  MoveL (T15717) to (119.32, 120.67, 17.1) mm, rotated rx 180 ry 0 rz -180 deg; joints [1.326, 66.029, -27.799, 2.142, -38.249, -1.682]
  Call Extruder 0.59936
  MoveL (T15718) to (105.47, 106.82, 17.1) mm, rotated rx 180 ry 0 rz -180 deg; joints [1.326, 66.029, -27.799, 2.142, -38.249, -1.682]
  Call Extruder 0.0152
  MoveL (T15719) to (105.47, 107.32, 17.1) mm, rotated rx 180 ry 0 rz -180 deg; joints [1.326, 66.029, -27.799, 2.142, -38.249, -1.682]
  Call Extruder 0.00328
  MoveL (T15720) to (105.49, 107.42, 17.1) mm, rotated rx 180 ry 0 rz -180 deg; joints [1.326, 66.029, -27.799, 2.142, -38.249, -1.682]
  Call Extruder 0.58584
  MoveL (T15721) to (119.03, 120.96, 17.1) mm, rotated rx 180 ry 0 rz -180 deg; joints [1.326, 66.029, -27.799, 2.142, -38.249, -1.682]
  Call Extruder 0.0086
  MoveL (T15722) to (118.83, 121.16, 17.1) mm, rotated rx 180 ry 0 rz -180 deg; joints [1.326, 66.029, -27.799, 2.142, -38.249, -1.682]
  Call Extruder 0.00554
  MoveL (T15723) to (118.65, 121.16, 17.1) mm, rotated rx 180 ry 0 rz -180 deg; joints [1.326, 66.029, -27.799, 2.142, -38.249, -1.682]
  Call Extruder 0.55945
  MoveL (T15724) to (105.72, 108.23, 17.1) mm, rotated rx 180 ry 0 rz -180 deg; joints [1.326, 66.029, -27.799, 2.142, -38.249, -1.682]
  Call Extruder 0.04056
  MoveL (T15725) to (106.33, 109.41, 17.1) mm, rotated rx 180 ry 0 rz -180 deg; joints [1.326, 66.029, -27.799, 2.142, -38.249, -1.682]
  Call Extruder 0.50836
  MoveL (T15726) to (118.07, 121.16, 17.1) mm, rotated rx 180 ry 0 rz -180 deg; joints [1.323, 66.013, -27.77, 2.137, -38.263, -1.678]
  Call Extruder 0.0177
  MoveL (T15727) to (117.49, 121.16, 17.1) mm, rotated rx 180 ry 0 rz -180 deg; joints [1.323, 66.013, -27.77, 2.137, -38.263, -1.678]
  Call Extruder 0.45726
  MoveL (T15728) to (106.93, 110.59, 17.1) mm, rotated rx 180 ry 0 rz -180 deg; joints [1.323, 66.013, -27.77, 2.137, -38.263, -1.678]
  Call Extruder 0.04056
  MoveL (T15729) to (107.53, 111.77, 17.1) mm, rotated rx 180 ry 0 rz -180 deg; joints [1.323, 66.013, -27.77, 2.137, -38.263, -1.678]
  Call Extruder 0.40616
  MoveL (T15730) to (116.92, 121.16, 17.1) mm, rotated rx 180 ry 0 rz -180 deg; joints [1.321, 66.248, -28.211, 2.143, -38.056, -1.688]
  Call Extruder 0.0177
  MoveL (T15731) to (116.34, 121.16, 17.1) mm, rotated rx 180 ry 0 rz -180 deg; joints [1.321, 66.248, -28.211, 2.143, -38.056, -1.688]
  Call Extruder 0.35507
  MoveL (T15732) to (108.13, 112.95, 17.1) mm, rotated rx 180 ry 0 rz -180 deg; joints [1.321, 66.248, -28.211, 2.143, -38.056, -1.688]
  Call Extruder 0.03441
  MoveL (T15733) to (108.64, 113.95, 17.1) mm, rotated rx 180 ry 0 rz -180 deg; joints [1.321, 66.248, -28.211, 2.143, -38.056, -1.688]
  Call Extruder 0.00268
  MoveL (T15734) to (108.56, 113.95, 17.1) mm, rotated rx 180 ry 0 rz -180 deg; joints [1.321, 66.248, -28.211, 2.143, -38.056, -1.688]
  Call Extruder 0.31171
  MoveL (T15735) to (115.76, 121.16, 17.1) mm, rotated rx 180 ry 0 rz -180 deg; joints [1.402, 70.427, -36.068, 2.484, -34.384, -2.05]
  Call Extruder 0.0177
  MoveL (T15736) to (115.18, 121.16, 17.1) mm, rotated rx 180 ry 0 rz -180 deg; joints [1.402, 70.427, -36.068, 2.484, -34.384, -2.05]
  Call Extruder 0.31171
  MoveL (T15737) to (107.98, 113.95, 17.1) mm, rotated rx 180 ry 0 rz -180 deg; joints [1.402, 70.427, -36.068, 2.484, -34.384, -2.05]
  Call Extruder 0.01315
  MoveL (T15738) to (107.55, 113.95, 17.1) mm, rotated rx 180 ry 0 rz -180 deg; joints [1.402, 70.427, -36.068, 2.484, -34.384, -2.05]
  Call Extruder 0.00328
  MoveL (T15739) to (107.46, 114.01, 17.1) mm, rotated rx 180 ry 0 rz -180 deg; joints [1.402, 70.427, -36.068, 2.484, -34.384, -2.05]
  Call Extruder 0.30914
  MoveL (T15740) to (114.6, 121.16, 17.1) mm, rotated rx 180 ry 0 rz -180 deg; joints [1.402, 70.427, -36.068, 2.484, -34.384, -2.05]
  Call Extruder 0.0177
  MoveL (T15741) to (114.02, 121.16, 17.1) mm, rotated rx 180 ry 0 rz -180 deg; joints [1.402, 70.427, -36.068, 2.484, -34.384, -2.05]
  Call Extruder 0.29663
  MoveL (T15742) to (107.17, 114.3, 17.1) mm, rotated rx 180 ry 0 rz -180 deg; joints [1.402, 70.427, -36.068, 2.484, -34.384, -2.05]
  Call Extruder 0.01252
  MoveL (T15743) to (106.88, 114.59, 17.1) mm, rotated rx 180 ry 0 rz -180 deg; joints [1.402, 70.427, -36.068, 2.484, -34.384, -2.05]
  Call Extruder 0.28411
  MoveL (T15744) to (113.44, 121.16, 17.1) mm, rotated rx 180 ry 0 rz -180 deg; joints [1.396, 71.177, -37.479, 2.515, -33.723, -2.092]
  Call Extruder 0.0177
  MoveL (T15745) to (112.87, 121.16, 17.1) mm, rotated rx 180 ry 0 rz -180 deg; joints [1.396, 71.177, -37.479, 2.515, -33.723, -2.092]
  Call Extruder 0.2716
  MoveL (T15746) to (106.59, 114.88, 17.1) mm, rotated rx 180 ry 0 rz -180 deg; joints [1.396, 71.177, -37.479, 2.515, -33.723, -2.092]
  Call Extruder 0.01252
  MoveL (T15747) to (106.3, 115.17, 17.1) mm, rotated rx 180 ry 0 rz -180 deg; joints [3.316, 66.49, -28.667, 5.398, -37.947, -4.261]
  Call Extruder 0.25908
  MoveL (T15748) to (112.29, 121.16, 17.1) mm, rotated rx 180 ry 0 rz -180 deg; joints [3.316, 66.49, -28.667, 5.398, -37.947, -4.261]
  Call Extruder 0.0177
  MoveL (T15749) to (111.71, 121.16, 17.1) mm, rotated rx 180 ry 0 rz -180 deg; joints [2.938, 66.441, -28.574, 4.78, -37.964, -3.772]
  Call Extruder 0.24657
  MoveL (T15750) to (106.01, 115.46, 17.1) mm, rotated rx 180 ry 0 rz -180 deg; joints [2.938, 66.441, -28.574, 4.78, -37.964, -3.772]
  Call Extruder 0.01252
  MoveL (T15751) to (105.72, 115.75, 17.1) mm, rotated rx 180 ry 0 rz -180 deg; joints [3.295, 67.406, -30.389, 5.461, -37.143, -4.358]
  Call Extruder 0.23405
  MoveL (T15752) to (111.13, 121.16, 17.1) mm, rotated rx 180 ry 0 rz -180 deg; joints [3.295, 67.406, -30.389, 5.461, -37.143, -4.358]
  Call Extruder 0.0177
  MoveL (T15753) to (110.55, 121.16, 17.1) mm, rotated rx 180 ry 0 rz -180 deg; joints [3.288, 67.704, -30.949, 5.483, -36.882, -4.391]
  Call Extruder 0.21634
  MoveL (T15754) to (105.55, 116.16, 17.1) mm, rotated rx 180 ry 0 rz -180 deg; joints [3.288, 67.704, -30.949, 5.483, -36.882, -4.391]
  Call Extruder 0.0177
  MoveL (T15755) to (105.55, 116.73, 17.1) mm, rotated rx 180 ry 0 rz -180 deg; joints [1.879, 71.218, -37.556, 3.388, -33.708, -2.819]
  Call Extruder 0.19131
  MoveL (T15756) to (109.97, 121.16, 17.1) mm, rotated rx 180 ry 0 rz -180 deg; joints [1.879, 71.218, -37.556, 3.388, -33.708, -2.819]
  Call Extruder 0.0177
  MoveL (T15757) to (109.4, 121.16, 17.1) mm, rotated rx 180 ry 0 rz -180 deg; joints [1.879, 71.218, -37.556, 3.388, -33.708, -2.819]
  Call Extruder 0.16628
  MoveL (T15758) to (105.55, 117.31, 17.1) mm, rotated rx 180 ry 0 rz -180 deg; joints [1.763, 71.207, -37.535, 3.177, -33.712, -2.644]
  Call Extruder 0.0177
  MoveL (T15759) to (105.55, 117.89, 17.1) mm, rotated rx 180 ry 0 rz -180 deg; joints [1.763, 71.207, -37.535, 3.177, -33.712, -2.644]
  Call Extruder 0.14125
  MoveL (T15760) to (108.82, 121.16, 17.1) mm, rotated rx 180 ry 0 rz -180 deg; joints [1.405, 70.111, -35.474, 2.471, -34.662, -2.033]
  Call Extruder 0.0177
  MoveL (T15761) to (108.24, 121.16, 17.1) mm, rotated rx 180 ry 0 rz -180 deg; joints [1.405, 70.111, -35.474, 2.471, -34.662, -2.033]
  Call Extruder 0.11622
  MoveL (T15762) to (105.55, 118.47, 17.1) mm, rotated rx 180 ry 0 rz -180 deg; joints [1.405, 70.111, -35.474, 2.471, -34.662, -2.033]
  Call Extruder 0.0177
  MoveL (T15763) to (105.55, 119.05, 17.1) mm, rotated rx 180 ry 0 rz -180 deg; joints [1.408, 69.782, -34.856, 2.458, -34.951, -2.015]
  Call Extruder 0.09119
  MoveL (T15764) to (107.66, 121.16, 17.1) mm, rotated rx 180 ry 0 rz -180 deg; joints [2.818, 66.427, -28.547, 4.584, -37.969, -3.616]
  Call Extruder 0.0177
  MoveL (T15765) to (107.08, 121.16, 17.1) mm, rotated rx 180 ry 0 rz -180 deg; joints [2.44, 66.386, -28.47, 3.966, -37.982, -3.128]
  Call Extruder 0.06616
  MoveL (T15766) to (105.55, 119.63, 17.1) mm, rotated rx 180 ry 0 rz -180 deg; joints [2.44, 66.386, -28.47, 3.966, -37.982, -3.128]
  Call Extruder 0.01683
  MoveL (T15767) to (105.55, 120.18, 17.1) mm, rotated rx 180 ry 0 rz -180 deg; joints [3.266, 68.664, -32.754, 5.557, -36.039, -4.499]
  Call Extruder 0.00161
  MoveL (T15768) to (105.57, 120.23, 17.1) mm, rotated rx 180 ry 0 rz -180 deg; joints [3.266, 68.664, -32.754, 5.557, -36.039, -4.499]
  Call Extruder 0.04818
  MoveL (T15769) to (106.69, 121.34, 17.1) mm, rotated rx 180 ry 0 rz -180 deg; joints [3.266, 68.664, -32.754, 5.557, -36.039, -4.499]
  Set speed (45.0 mm/s)
  Call Extruder -1.6
  MoveL (T15770) to (106.69, 121.34, 17.1) mm, rotated rx 180 ry 0 rz -180 deg; joints [3.266, 68.664, -32.754, 5.557, -36.039, -4.499]
  Set speed (120.0 mm/s)
  MoveL (T15771) to (106.69, 121.34, 17.1) mm, rotated rx 180 ry 0 rz -180 deg; joints [3.26, 68.978, -33.343, 5.583, -35.764, -4.535]
  Call Extruder -0.38
  MoveL (T15772) to (105.93, 120.58, 17.1) mm, rotated rx 180 ry 0 rz -180 deg; joints [3.26, 68.978, -33.343, 5.583, -35.764, -4.535]
  Set speed (45.0 mm/s)
  Call Extruder -0.02
  MoveL (T15773) to (105.93, 120.58, 17.1) mm, rotated rx 180 ry 0 rz -180 deg; joints [3.26, 68.978, -33.343, 5.583, -35.764, -4.535]
  Set speed (150.0 mm/s)
  MoveL (T15774) to (105.93, 120.58, 19.1) mm, rotated rx 180 ry 0 rz -180 deg; joints [2.362, 71.271, -37.657, 4.262, -33.688, -3.548]
  MoveL (T15775) to (120.54, 120.54, 19.1) mm, rotated rx 180 ry 0 rz -180 deg; joints [2.362, 71.271, -37.657, 4.262, -33.688, -3.548]
  MoveL (T15776) to (120.54, 120.54, 17.1) mm, rotated rx 180 ry 0 rz -180 deg; joints [2.362, 71.271, -37.657, 4.262, -33.688, -3.548]
  Set speed (40.0 mm/s)
  Call Extruder 2.0
  MoveL (T15777) to (120.54, 120.54, 17.1) mm, rotated rx 180 ry 0 rz -180 deg; joints [2.246, 71.257, -37.63, 4.051, -33.693, -3.372]
  Set speed (50.0 mm/s)
  MoveL (T15778) to (120.54, 120.54, 17.1) mm, rotated rx 180 ry 0 rz -180 deg; joints [2.246, 71.257, -37.63, 4.051, -33.693, -3.372]
  Call Extruder 0.02637
  MoveL (T15779) to (121.16, 121.16, 17.1) mm, rotated rx 180 ry 0 rz -180 deg; joints [2.246, 71.257, -37.63, 4.051, -33.693, -3.372]
  Set speed (45.0 mm/s)
  Call Extruder -1.6
  MoveL (T15780) to (121.16, 121.16, 17.1) mm, rotated rx 180 ry 0 rz -180 deg; joints [1.417, 68.778, -32.967, 2.421, -35.835, -1.963]
  Set speed (120.0 mm/s)
  MoveL (T15781) to (121.16, 121.16, 17.1) mm, rotated rx 180 ry 0 rz -180 deg; joints [1.417, 68.778, -32.967, 2.421, -35.835, -1.963]
  Call Extruder -0.30841
  MoveL (T15782) to (120.54, 120.54, 17.1) mm, rotated rx 180 ry 0 rz -180 deg; joints [1.42, 68.466, -32.382, 2.41, -36.109, -1.947]
  Set speed (45.0 mm/s)
  Call Extruder -0.09159
  MoveL (T15783) to (120.54, 120.54, 17.1) mm, rotated rx 180 ry 0 rz -180 deg; joints [1.42, 68.466, -32.382, 2.41, -36.109, -1.947]
  Set speed (150.0 mm/s)
  MoveL (T15784) to (120.54, 120.54, 19.1) mm, rotated rx 180 ry 0 rz -180 deg; joints [1.42, 68.466, -32.382, 2.41, -36.109, -1.947]
  MoveL (T15785) to (104.34, 103.54, 19.1) mm, rotated rx 180 ry 0 rz -180 deg; joints [1.42, 68.466, -32.382, 2.41, -36.109, -1.947]
  MoveL (T15786) to (104.34, 103.54, 17.3) mm, rotated rx 180 ry 0 rz -180 deg; joints [2.319, 66.374, -28.448, 3.77, -37.986, -2.973]
  Set speed (40.0 mm/s)
  Call Extruder 2.0
  MoveL (T15787) to (104.34, 103.54, 17.3) mm, rotated rx 180 ry 0 rz -180 deg; joints [2.319, 66.374, -28.448, 3.77, -37.986, -2.973]
  Call Extruder 0.52159
  MoveL (T15788) to (121.46, 103.54, 17.3) mm, rotated rx 180 ry 0 rz -180 deg; joints [2.319, 66.374, -28.448, 3.77, -37.986, -2.973]
  Call Extruder 0.54596
  MoveL (T15789) to (121.46, 121.46, 17.3) mm, rotated rx 180 ry 0 rz -180 deg; joints [2.319, 66.374, -28.448, 3.77, -37.986, -2.973]
  Call Extruder 0.54596
  MoveL (T15790) to (103.54, 121.46, 17.3) mm, rotated rx 180 ry 0 rz -180 deg; joints [1.941, 66.34, -28.385, 3.154, -37.998, -2.486]
  Call Extruder 0.54596
  MoveL (T15791) to (103.54, 103.54, 17.3) mm, rotated rx 180 ry 0 rz -180 deg; joints [1.941, 66.34, -28.385, 3.154, -37.998, -2.486]
  Call Extruder 0.02254
  MoveL (T15792) to (104.28, 103.54, 17.3) mm, rotated rx 180 ry 0 rz -180 deg; joints [1.941, 66.34, -28.385, 3.154, -37.998, -2.486]
  Set speed (150.0 mm/s)
  MoveL (T15793) to (103.53, 103.13, 17.3) mm, rotated rx 180 ry 0 rz -180 deg; joints [3.239, 69.99, -35.246, 5.67, -34.875, -4.657]
  Set speed (40.0 mm/s)
  MoveL (T15794) to (103.53, 103.13, 17.3) mm, rotated rx 180 ry 0 rz -180 deg; joints [3.239, 69.99, -35.246, 5.67, -34.875, -4.657]
  Call Extruder 0.55858
  MoveL (T15795) to (121.87, 103.13, 17.3) mm, rotated rx 180 ry 0 rz -180 deg; joints [3.239, 69.99, -35.246, 5.67, -34.875, -4.657]
  Call Extruder 0.57077
  MoveL (T15796) to (121.87, 121.87, 17.3) mm, rotated rx 180 ry 0 rz -180 deg; joints [3.232, 70.321, -35.869, 5.7, -34.585, -4.698]
  Call Extruder 0.57077
  MoveL (T15797) to (103.13, 121.87, 17.3) mm, rotated rx 180 ry 0 rz -180 deg; joints [3.232, 70.321, -35.869, 5.7, -34.585, -4.698]
  Call Extruder 0.57077
  MoveL (T15798) to (103.13, 103.13, 17.3) mm, rotated rx 180 ry 0 rz -180 deg; joints [2.845, 71.337, -37.78, 5.138, -33.663, -4.28]
  Call Extruder 0.01036
  MoveL (T15799) to (103.47, 103.13, 17.3) mm, rotated rx 180 ry 0 rz -180 deg; joints [2.845, 71.337, -37.78, 5.138, -33.663, -4.28]
  Set speed (150.0 mm/s)
  MoveL (T15800) to (102.72, 102.81, 17.3) mm, rotated rx 180 ry 0 rz -180 deg; joints [2.729, 71.32, -37.748, 4.926, -33.669, -4.103]
  Set speed (25.0 mm/s)
  MoveL (T15801) to (102.72, 102.81, 17.3) mm, rotated rx 180 ry 0 rz -180 deg; joints [2.729, 71.32, -37.748, 4.926, -33.669, -4.103]
  Call Extruder 0.00259
  MoveL (T15802) to (102.72, 102.72, 17.3) mm, rotated rx 180 ry 0 rz -180 deg; joints [2.729, 71.32, -37.748, 4.926, -33.669, -4.103]
  Call Extruder 0.59557
  MoveL (T15803) to (122.28, 102.72, 17.3) mm, rotated rx 180 ry 0 rz -180 deg; joints [1.429, 67.513, -30.588, 2.378, -36.948, -1.901]
  Call Extruder 0.59557
  MoveL (T15804) to (122.28, 122.28, 17.3) mm, rotated rx 180 ry 0 rz -180 deg; joints [1.429, 67.513, -30.588, 2.378, -36.948, -1.901]
  Call Extruder 0.59557
  MoveL (T15805) to (102.72, 122.28, 17.3) mm, rotated rx 180 ry 0 rz -180 deg; joints [1.429, 67.513, -30.588, 2.378, -36.948, -1.901]
  Call Extruder 0.59115
  MoveL (T15806) to (102.72, 102.87, 17.3) mm, rotated rx 180 ry 0 rz -180 deg; joints [1.432, 67.216, -30.031, 2.369, -37.209, -1.887]
  Set speed (150.0 mm/s)
  MoveL (T15807) to (102.78, 102.75, 17.3) mm, rotated rx 180 ry 0 rz -180 deg; joints [1.432, 67.216, -30.031, 2.369, -37.209, -1.887]
  Set speed (45.0 mm/s)
  Call Extruder -1.6
  MoveL (T15808) to (102.78, 102.75, 17.3) mm, rotated rx 180 ry 0 rz -180 deg; joints [1.821, 66.331, -28.367, 2.958, -38.001, -2.332]
  Set speed (120.0 mm/s)
  MoveL (T15809) to (102.78, 102.75, 17.3) mm, rotated rx 180 ry 0 rz -180 deg; joints [1.821, 66.331, -28.367, 2.958, -38.001, -2.332]
  Call Extruder -0.05166
  MoveL (T15810) to (102.72, 102.72, 17.3) mm, rotated rx 180 ry 0 rz -180 deg; joints [1.821, 66.331, -28.367, 2.958, -38.001, -2.332]
  Call Extruder -0.32834
  MoveL (T15811) to (103.65, 102.72, 17.3) mm, rotated rx 180 ry 0 rz -180 deg; joints [1.442, 66.306, -28.319, 2.342, -38.01, -1.845]
  Set speed (45.0 mm/s)
  Call Extruder -0.02
  MoveL (T15812) to (103.65, 102.72, 17.3) mm, rotated rx 180 ry 0 rz -180 deg; joints [1.442, 66.306, -28.319, 2.342, -38.01, -1.845]
  Set speed (150.0 mm/s)
  MoveL (T15813) to (103.65, 102.72, 19.3) mm, rotated rx 180 ry 0 rz -180 deg; joints [1.442, 66.306, -28.319, 2.342, -38.01, -1.845]
  MoveL (T15814) to (106.08, 103.93, 19.3) mm, rotated rx 180 ry 0 rz -180 deg; joints [1.442, 66.306, -28.319, 2.342, -38.01, -1.845]
  MoveL (T15815) to (106.08, 103.93, 17.3) mm, rotated rx 180 ry 0 rz -180 deg; joints [3.211, 71.395, -37.89, 5.803, -33.641, -4.837]
  Set speed (40.0 mm/s)
  Call Extruder 2.0
  MoveL (T15816) to (106.08, 103.93, 17.3) mm, rotated rx 180 ry 0 rz -180 deg; joints [3.211, 71.395, -37.89, 5.803, -33.641, -4.837]
  Set speed (50.0 mm/s)
  MoveL (T15817) to (106.08, 103.93, 17.3) mm, rotated rx 180 ry 0 rz -180 deg; joints [3.211, 71.395, -37.89, 5.803, -33.641, -4.837]
  Call Extruder 0.00361
  MoveL (T15818) to (106.17, 103.84, 17.3) mm, rotated rx 180 ry 0 rz -180 deg; joints [3.226, 70.639, -36.467, 5.73, -34.305, -4.738]
  Call Extruder 0.0708
  MoveL (T15819) to (103.84, 103.84, 17.3) mm, rotated rx 180 ry 0 rz -180 deg; joints [3.226, 70.639, -36.467, 5.73, -34.305, -4.738]
  Call Extruder 0.05255
  MoveL (T15820) to (105.06, 105.06, 17.3) mm, rotated rx 180 ry 0 rz -180 deg; joints [3.226, 70.639, -36.467, 5.73, -34.305, -4.738]
  Call Extruder 0.03217
  MoveL (T15821) to (105.06, 106.12, 17.3) mm, rotated rx 180 ry 0 rz -180 deg; joints [3.226, 70.639, -36.467, 5.73, -34.305, -4.738]
  Call Extruder 0.0525
  MoveL (T15822) to (103.84, 107.34, 17.3) mm, rotated rx 180 ry 0 rz -180 deg; joints [3.226, 70.639, -36.467, 5.73, -34.305, -4.738]
  Call Extruder 0.03385
  MoveL (T15823) to (103.84, 108.45, 17.3) mm, rotated rx 180 ry 0 rz -180 deg; joints [3.226, 70.639, -36.467, 5.73, -34.305, -4.738]
  Call Extruder 0.13495
  MoveL (T15824) to (106.98, 111.58, 17.3) mm, rotated rx 180 ry 0 rz -180 deg; joints [3.226, 70.639, -36.467, 5.73, -34.305, -4.738]
  Call Extruder 0.04156
  MoveL (T15825) to (107.6, 112.8, 17.3) mm, rotated rx 180 ry 0 rz -180 deg; joints [3.226, 70.639, -36.467, 5.73, -34.305, -4.738]
  Call Extruder 0.16166
  MoveL (T15826) to (103.84, 116.55, 17.3) mm, rotated rx 180 ry 0 rz -180 deg; joints [3.226, 70.639, -36.467, 5.73, -34.305, -4.738]
  Call Extruder 0.03385
  MoveL (T15827) to (103.84, 117.66, 17.3) mm, rotated rx 180 ry 0 rz -180 deg; joints [3.226, 70.639, -36.467, 5.73, -34.305, -4.738]
  Call Extruder 0.05612
  MoveL (T15828) to (105.15, 118.96, 17.3) mm, rotated rx 180 ry 0 rz -180 deg; joints [3.226, 70.639, -36.467, 5.73, -34.305, -4.738]
  Call Extruder 0.02709
  MoveL (T15829) to (105.15, 119.85, 17.3) mm, rotated rx 180 ry 0 rz -180 deg; joints [3.226, 70.639, -36.467, 5.73, -34.305, -4.738]
  Call Extruder 0.05612
  MoveL (T15830) to (103.84, 121.16, 17.3) mm, rotated rx 180 ry 0 rz -180 deg; joints [3.219, 70.966, -37.082, 5.761, -34.018, -4.78]
  Call Extruder 0.06345
  MoveL (T15831) to (105.93, 121.16, 17.3) mm, rotated rx 180 ry 0 rz -180 deg; joints [3.219, 70.966, -37.082, 5.761, -34.018, -4.78]
  Call Extruder 0.01096
  MoveL (T15832) to (105.67, 120.9, 17.3) mm, rotated rx 180 ry 0 rz -180 deg; joints [3.219, 70.966, -37.082, 5.761, -34.018, -4.78]
  Set speed (45.0 mm/s)
  Call Extruder -1.6
  MoveL (T15833) to (105.67, 120.9, 17.3) mm, rotated rx 180 ry 0 rz -180 deg; joints [3.219, 70.966, -37.082, 5.761, -34.018, -4.78]
  Set speed (120.0 mm/s)
  MoveL (T15834) to (105.67, 120.9, 17.3) mm, rotated rx 180 ry 0 rz -180 deg; joints [3.219, 70.966, -37.082, 5.761, -34.018, -4.78]
  Call Extruder -0.12811
  MoveL (T15835) to (105.93, 121.16, 17.3) mm, rotated rx 180 ry 0 rz -180 deg; joints [3.219, 70.966, -37.082, 5.761, -34.018, -4.78]
  Call Extruder -0.25189
  MoveL (T15836) to (105.22, 121.16, 17.3) mm, rotated rx 180 ry 0 rz -180 deg; joints [3.219, 70.732, -37.037, 5.789, -33.83, -4.814]
  Set speed (45.0 mm/s)
  Call Extruder -0.02
  MoveL (T15837) to (105.22, 121.16, 17.3) mm, rotated rx 180 ry 0 rz -180 deg; joints [1.407, 66.407, -28.551, 2.292, -37.879, -1.81]
  Set speed (150.0 mm/s)
  MoveL (T15838) to (105.22, 121.16, 19.3) mm, rotated rx 180 ry 0 rz -180 deg; joints [1.407, 66.407, -28.551, 2.292, -37.879, -1.81]
  MoveL (T15839) to (105.15, 117.23, 19.3) mm, rotated rx 180 ry 0 rz -180 deg; joints [1.407, 66.407, -28.551, 2.292, -37.879, -1.81]
  MoveL (T15840) to (105.15, 117.23, 17.3) mm, rotated rx 180 ry 0 rz -180 deg; joints [1.407, 66.407, -28.551, 2.292, -37.879, -1.81]
  Set speed (40.0 mm/s)
  Call Extruder 2.0
  MoveL (T15841) to (105.15, 117.23, 17.3) mm, rotated rx 180 ry 0 rz -180 deg; joints [1.407, 66.407, -28.551, 2.292, -37.879, -1.81]
  Set speed (50.0 mm/s)
  MoveL (T15842) to (105.15, 117.23, 17.3) mm, rotated rx 180 ry 0 rz -180 deg; joints [1.407, 66.407, -28.551, 2.292, -37.879, -1.81]
  Call Extruder 0.04143
  MoveL (T15843) to (105.15, 115.87, 17.3) mm, rotated rx 180 ry 0 rz -180 deg; joints [1.407, 66.407, -28.551, 2.292, -37.879, -1.81]
  Call Extruder 0.00661
  MoveL (T15844) to (105.23, 115.67, 17.3) mm, rotated rx 180 ry 0 rz -180 deg; joints [1.407, 66.407, -28.551, 2.292, -37.879, -1.81]
  Call Extruder 0.02637
  MoveL (T15845) to (105.84, 115.05, 17.3) mm, rotated rx 180 ry 0 rz -180 deg; joints [1.407, 66.407, -28.551, 2.292, -37.879, -1.81]
  Call Extruder 0.08606
  MoveL (T15846) to (103.84, 113.06, 17.3) mm, rotated rx 180 ry 0 rz -180 deg; joints [1.407, 66.407, -28.551, 2.292, -37.879, -1.81]
  Call Extruder 0.03385
  MoveL (T15847) to (103.84, 111.94, 17.3) mm, rotated rx 180 ry 0 rz -180 deg; joints [1.363, 71.246, -37.649, 2.462, -33.622, -2.051]
  Call Extruder 0.09463
  MoveL (T15848) to (106.04, 109.75, 17.3) mm, rotated rx 180 ry 0 rz -180 deg; joints [3.241, 71.473, -38.076, 5.874, -33.536, -4.902]
  Call Extruder 0.05062
  MoveL (T15849) to (105.29, 108.27, 17.3) mm, rotated rx 180 ry 0 rz -180 deg; joints [3.241, 71.473, -38.076, 5.874, -33.536, -4.902]
  Call Extruder 0.02377
  MoveL (T15850) to (105.1, 107.51, 17.3) mm, rotated rx 180 ry 0 rz -180 deg; joints [3.241, 71.473, -38.076, 5.874, -33.536, -4.902]
  Set speed (45.0 mm/s)
  Call Extruder -1.6
  MoveL (T15851) to (105.1, 107.51, 17.3) mm, rotated rx 180 ry 0 rz -180 deg; joints [3.351, 66.393, -28.524, 5.449, -37.995, -4.299]
  Set speed (120.0 mm/s)
  MoveL (T15852) to (105.1, 107.51, 17.3) mm, rotated rx 180 ry 0 rz -180 deg; joints [3.351, 66.393, -28.524, 5.449, -37.995, -4.299]
  Call Extruder -0.278
  MoveL (T15853) to (105.29, 108.27, 17.3) mm, rotated rx 180 ry 0 rz -180 deg; joints [1.409, 66.202, -28.165, 2.287, -38.059, -1.801]
  Call Extruder -0.102
  MoveL (T15854) to (105.42, 108.52, 17.3) mm, rotated rx 180 ry 0 rz -180 deg; joints [1.409, 66.202, -28.165, 2.287, -38.059, -1.801]
  Set speed (45.0 mm/s)
  Call Extruder -0.02
  MoveL (T15855) to (105.42, 108.52, 17.3) mm, rotated rx 180 ry 0 rz -180 deg; joints [1.409, 66.202, -28.165, 2.287, -38.059, -1.801]
  Set speed (150.0 mm/s)
  MoveL (T15856) to (105.42, 108.52, 19.3) mm, rotated rx 180 ry 0 rz -180 deg; joints [1.407, 66.392, -28.522, 2.292, -37.892, -1.809]
  MoveL (T15857) to (119.44, 110.51, 19.3) mm, rotated rx 180 ry 0 rz -180 deg; joints [1.407, 66.392, -28.522, 2.292, -37.892, -1.809]
  MoveL (T15858) to (119.44, 110.51, 17.3) mm, rotated rx 180 ry 0 rz -180 deg; joints [1.365, 66.197, -28.157, 2.215, -38.061, -1.744]
  Set speed (40.0 mm/s)
  Call Extruder 2.0
  MoveL (T15859) to (119.44, 110.51, 17.3) mm, rotated rx 180 ry 0 rz -180 deg; joints [1.365, 66.197, -28.157, 2.215, -38.061, -1.744]
  Set speed (50.0 mm/s)
  MoveL (T15860) to (119.44, 110.51, 17.3) mm, rotated rx 180 ry 0 rz -180 deg; joints [1.365, 66.197, -28.157, 2.215, -38.061, -1.744]
  Call Extruder 0.05098
  MoveL (T15861) to (118.25, 111.7, 17.3) mm, rotated rx 180 ry 0 rz -180 deg; joints [1.365, 66.197, -28.157, 2.215, -38.061, -1.744]
  Call Extruder 0.00661
  MoveL (T15862) to (118.05, 111.78, 17.3) mm, rotated rx 180 ry 0 rz -180 deg; joints [1.319, 71.371, -37.884, 2.391, -33.51, -1.994]
  Call Extruder 0.00686
  MoveL (T15863) to (117.83, 111.78, 17.3) mm, rotated rx 180 ry 0 rz -180 deg; joints [1.319, 71.371, -37.884, 2.391, -33.51, -1.994]
  Call Extruder 0.01607
  MoveL (T15864) to (117.45, 112.15, 17.3) mm, rotated rx 180 ry 0 rz -180 deg; joints [1.319, 71.371, -37.884, 2.391, -33.51, -1.994]
  Call Extruder 0.04881
  MoveL (T15865) to (118.18, 113.58, 17.3) mm, rotated rx 180 ry 0 rz -180 deg; joints [1.319, 71.371, -37.884, 2.391, -33.51, -1.994]
  Call Extruder 0.12804
  MoveL (T15866) to (121.16, 116.55, 17.3) mm, rotated rx 180 ry 0 rz -180 deg; joints [1.319, 71.371, -37.884, 2.391, -33.51, -1.994]
  Call Extruder 0.03385
  MoveL (T15867) to (121.16, 117.66, 17.3) mm, rotated rx 180 ry 0 rz -180 deg; joints [3.282, 71.61, -38.333, 5.966, -33.42, -4.985]
  Call Extruder 0.04175
  MoveL (T15868) to (120.19, 118.63, 17.3) mm, rotated rx 180 ry 0 rz -180 deg; joints [3.282, 71.61, -38.333, 5.966, -33.42, -4.985]
  Call Extruder 0.04741
  MoveL (T15869) to (120.19, 120.19, 17.3) mm, rotated rx 180 ry 0 rz -180 deg; joints [3.282, 71.61, -38.333, 5.966, -33.42, -4.985]
  Call Extruder 0.04175
  MoveL (T15870) to (121.16, 121.16, 17.3) mm, rotated rx 180 ry 0 rz -180 deg; joints [3.282, 71.61, -38.333, 5.966, -33.42, -4.985]
  Call Extruder 0.07441
  MoveL (T15871) to (121.16, 118.71, 17.3) mm, rotated rx 180 ry 0 rz -180 deg; joints [3.398, 66.294, -28.339, 5.514, -38.084, -4.345]
  Set speed (150.0 mm/s)
  MoveL (T15872) to (120.05, 117.4, 17.3) mm, rotated rx 180 ry 0 rz -180 deg; joints [3.398, 66.294, -28.339, 5.514, -38.084, -4.345]
  Set speed (50.0 mm/s)
  MoveL (T15873) to (120.05, 117.4, 17.3) mm, rotated rx 180 ry 0 rz -180 deg; joints [1.366, 66.095, -27.965, 2.212, -38.151, -1.74]
  Call Extruder 0.01089
  MoveL (T15874) to (119.96, 117.05, 17.3) mm, rotated rx 180 ry 0 rz -180 deg; joints [1.366, 66.095, -27.965, 2.212, -38.151, -1.74]
  Call Extruder 0.0635
  MoveL (T15875) to (119.01, 115.2, 17.3) mm, rotated rx 180 ry 0 rz -180 deg; joints [1.366, 66.095, -27.965, 2.212, -38.151, -1.74]
  Call Extruder 0.09231
  MoveL (T15876) to (121.16, 113.06, 17.3) mm, rotated rx 180 ry 0 rz -180 deg; joints [1.365, 66.182, -28.128, 2.215, -38.075, -1.744]
  Call Extruder 0.03385
  MoveL (T15877) to (121.16, 111.94, 17.3) mm, rotated rx 180 ry 0 rz -180 deg; joints [1.365, 66.182, -28.128, 2.215, -38.075, -1.744]
  Call Extruder 0.06789
  MoveL (T15878) to (119.58, 110.37, 17.3) mm, rotated rx 180 ry 0 rz -180 deg; joints [1.332, 65.99, -27.767, 2.153, -38.243, -1.691]
  Call Extruder 0.03053
  MoveL (T15879) to (120.29, 109.66, 17.3) mm, rotated rx 180 ry 0 rz -180 deg; joints [1.332, 65.99, -27.767, 2.153, -38.243, -1.691]
  Call Extruder 0.00661
  MoveL (T15880) to (120.37, 109.46, 17.3) mm, rotated rx 180 ry 0 rz -180 deg; joints [1.332, 65.99, -27.767, 2.153, -38.243, -1.691]
  Call Extruder 0.00686
  MoveL (T15881) to (120.37, 109.23, 17.3) mm, rotated rx 180 ry 0 rz -180 deg; joints [1.323, 65.989, -27.766, 2.138, -38.243, -1.679]
  Call Extruder 0.03378
  MoveL (T15882) to (121.16, 108.45, 17.3) mm, rotated rx 180 ry 0 rz -180 deg; joints [1.323, 65.989, -27.766, 2.138, -38.243, -1.679]
  Call Extruder 0.03385
  MoveL (T15883) to (121.16, 107.34, 17.3) mm, rotated rx 180 ry 0 rz -180 deg; joints [1.276, 71.497, -38.121, 2.318, -33.398, -1.936]
  Call Extruder 0.03378
  MoveL (T15884) to (120.37, 106.56, 17.3) mm, rotated rx 180 ry 0 rz -180 deg; joints [1.276, 71.497, -38.121, 2.318, -33.398, -1.936]
  Call Extruder 0.04531
  MoveL (T15885) to (120.37, 105.07, 17.3) mm, rotated rx 180 ry 0 rz -180 deg; joints [1.276, 71.497, -38.121, 2.318, -33.398, -1.936]
  Call Extruder 0.00661
  MoveL (T15886) to (120.29, 104.87, 17.3) mm, rotated rx 180 ry 0 rz -180 deg; joints [1.276, 71.497, -38.121, 2.318, -33.398, -1.936]
  Call Extruder 0.00334
  MoveL (T15887) to (120.21, 104.79, 17.3) mm, rotated rx 180 ry 0 rz -180 deg; joints [3.322, 71.747, -38.592, 6.057, -33.303, -5.068]
  Call Extruder 0.04071
  MoveL (T15888) to (121.16, 103.84, 17.3) mm, rotated rx 180 ry 0 rz -180 deg; joints [3.322, 71.747, -38.592, 6.057, -33.303, -5.068]
  Call Extruder 0.07441
  MoveL (T15889) to (121.16, 106.29, 17.3) mm, rotated rx 180 ry 0 rz -180 deg; joints [3.322, 71.747, -38.592, 6.057, -33.303, -5.068]
  Set speed (45.0 mm/s)
  Call Extruder -1.6
  MoveL (T15890) to (121.16, 106.29, 17.3) mm, rotated rx 180 ry 0 rz -180 deg; joints [3.445, 66.197, -28.155, 5.579, -38.173, -4.391]
  Set speed (120.0 mm/s)
  MoveL (T15891) to (121.16, 106.29, 17.3) mm, rotated rx 180 ry 0 rz -180 deg; joints [1.339, 65.99, -27.768, 2.163, -38.243, -1.699]
  Call Extruder -0.38
  MoveL (T15892) to (121.16, 105.22, 17.3) mm, rotated rx 180 ry 0 rz -180 deg; joints [1.339, 65.99, -27.768, 2.163, -38.243, -1.699]
  Set speed (45.0 mm/s)
  Call Extruder -0.02
  MoveL (T15893) to (121.16, 105.22, 17.3) mm, rotated rx 180 ry 0 rz -180 deg; joints [1.339, 65.99, -27.768, 2.163, -38.243, -1.699]
  Set speed (150.0 mm/s)
  MoveL (T15894) to (121.16, 105.22, 19.3) mm, rotated rx 180 ry 0 rz -180 deg; joints [1.326, 66.005, -27.795, 2.143, -38.229, -1.683]
  MoveL (T15895) to (120.15, 108.89, 19.3) mm, rotated rx 180 ry 0 rz -180 deg; joints [1.326, 66.005, -27.795, 2.143, -38.229, -1.683]
  MoveL (T15896) to (120.15, 108.89, 17.3) mm, rotated rx 180 ry 0 rz -180 deg; joints [1.326, 66.005, -27.795, 2.143, -38.229, -1.683]
  Set speed (40.0 mm/s)
  Call Extruder 2.0
  MoveL (T15897) to (120.15, 108.89, 17.3) mm, rotated rx 180 ry 0 rz -180 deg; joints [1.326, 66.005, -27.795, 2.143, -38.229, -1.683]
  Call Extruder 0.11511
  MoveL (T15898) to (117.48, 111.56, 17.3) mm, rotated rx 180 ry 0 rz -180 deg; joints [1.326, 66.005, -27.795, 2.143, -38.229, -1.683]
  Set speed (45.0 mm/s)
  Call Extruder -1.6
  MoveL (T15899) to (117.48, 111.56, 17.3) mm, rotated rx 180 ry 0 rz -180 deg; joints [1.326, 66.005, -27.795, 2.143, -38.229, -1.683]
  Set speed (120.0 mm/s)
  MoveL (T15900) to (117.48, 111.56, 17.3) mm, rotated rx 180 ry 0 rz -180 deg; joints [1.326, 66.005, -27.795, 2.143, -38.229, -1.683]
  Call Extruder -0.38
  MoveL (T15901) to (118.23, 110.8, 17.3) mm, rotated rx 180 ry 0 rz -180 deg; joints [1.326, 66.005, -27.795, 2.143, -38.229, -1.683]
  Set speed (45.0 mm/s)
  Call Extruder -0.02
  MoveL (T15902) to (118.23, 110.8, 17.3) mm, rotated rx 180 ry 0 rz -180 deg; joints [1.326, 66.005, -27.795, 2.143, -38.229, -1.683]
  Set speed (150.0 mm/s)
  MoveL (T15903) to (118.23, 110.8, 19.3) mm, rotated rx 180 ry 0 rz -180 deg; joints [1.326, 66.005, -27.795, 2.143, -38.229, -1.683]
  MoveL (T15904) to (118.65, 121.34, 19.3) mm, rotated rx 180 ry 0 rz -180 deg; joints [1.326, 66.005, -27.795, 2.143, -38.229, -1.683]
  MoveL (T15905) to (118.65, 121.34, 17.3) mm, rotated rx 180 ry 0 rz -180 deg; joints [1.323, 65.989, -27.766, 2.138, -38.243, -1.679]
  Set speed (40.0 mm/s)
  Call Extruder 2.0
  MoveL (T15906) to (118.65, 121.34, 17.3) mm, rotated rx 180 ry 0 rz -180 deg; joints [1.323, 65.989, -27.766, 2.138, -38.243, -1.679]
  Call Extruder 0.04796
  MoveL (T15907) to (119.76, 120.23, 17.3) mm, rotated rx 180 ry 0 rz -180 deg; joints [1.321, 66.224, -28.207, 2.144, -38.036, -1.689]
  Call Extruder 0.00166
  MoveL (T15908) to (119.78, 120.18, 17.3) mm, rotated rx 180 ry 0 rz -180 deg; joints [1.321, 66.224, -28.207, 2.144, -38.036, -1.689]
  Call Extruder 0.01669
  MoveL (T15909) to (119.78, 119.63, 17.3) mm, rotated rx 180 ry 0 rz -180 deg; joints [1.321, 66.224, -28.207, 2.144, -38.036, -1.689]
  Call Extruder 0.06581
  MoveL (T15910) to (118.25, 121.16, 17.3) mm, rotated rx 180 ry 0 rz -180 deg; joints [1.321, 66.224, -28.207, 2.144, -38.036, -1.689]
  Call Extruder 0.01758
  MoveL (T15911) to (117.68, 121.16, 17.3) mm, rotated rx 180 ry 0 rz -180 deg; joints [1.321, 66.224, -28.207, 2.144, -38.036, -1.689]
  Call Extruder 0.09068
  MoveL (T15912) to (119.78, 119.05, 17.3) mm, rotated rx 180 ry 0 rz -180 deg; joints [1.321, 66.224, -28.207, 2.144, -38.036, -1.689]
  Call Extruder 0.01758
  MoveL (T15913) to (119.78, 118.48, 17.3) mm, rotated rx 180 ry 0 rz -180 deg; joints [1.402, 70.169, -36.019, 2.497, -34.175, -2.066]
  Call Extruder 0.11554
  MoveL (T15914) to (117.1, 121.16, 17.3) mm, rotated rx 180 ry 0 rz -180 deg; joints [1.402, 70.403, -36.063, 2.485, -34.365, -2.051]
  Call Extruder 0.01758
  MoveL (T15915) to (116.52, 121.16, 17.3) mm, rotated rx 180 ry 0 rz -180 deg; joints [1.402, 70.403, -36.063, 2.485, -34.365, -2.051]
  Call Extruder 0.13957
  MoveL (T15916) to (119.76, 117.92, 17.3) mm, rotated rx 180 ry 0 rz -180 deg; joints [1.402, 70.403, -36.063, 2.485, -34.365, -2.051]
  Call Extruder 0.01457
  MoveL (T15917) to (119.65, 117.45, 17.3) mm, rotated rx 180 ry 0 rz -180 deg; joints [1.402, 70.403, -36.063, 2.485, -34.365, -2.051]
  Call Extruder 0.15961
  MoveL (T15918) to (115.95, 121.16, 17.3) mm, rotated rx 180 ry 0 rz -180 deg; joints [1.402, 70.403, -36.063, 2.485, -34.365, -2.051]
  Call Extruder 0.01758
  MoveL (T15919) to (115.37, 121.16, 17.3) mm, rotated rx 180 ry 0 rz -180 deg; joints [1.402, 70.403, -36.063, 2.485, -34.365, -2.051]
  Call Extruder 0.17783
  MoveL (T15920) to (119.49, 117.03, 17.3) mm, rotated rx 180 ry 0 rz -180 deg; joints [1.402, 70.403, -36.063, 2.485, -34.365, -2.051]
  Call Extruder 0.01306
  MoveL (T15921) to (119.3, 116.65, 17.3) mm, rotated rx 180 ry 0 rz -180 deg; joints [1.402, 70.403, -36.063, 2.485, -34.365, -2.051]
  Call Extruder 0.19428
  MoveL (T15922) to (114.8, 121.16, 17.3) mm, rotated rx 180 ry 0 rz -180 deg; joints [1.402, 70.403, -36.063, 2.485, -34.365, -2.051]
  Call Extruder 0.01758
  MoveL (T15923) to (114.22, 121.16, 17.3) mm, rotated rx 180 ry 0 rz -180 deg; joints [1.402, 70.403, -36.063, 2.485, -34.365, -2.051]
  Call Extruder 0.21073
  MoveL (T15924) to (119.1, 116.27, 17.3) mm, rotated rx 180 ry 0 rz -180 deg; joints [1.402, 70.403, -36.063, 2.485, -34.365, -2.051]
  Call Extruder 0.01306
  MoveL (T15925) to (118.91, 115.89, 17.3) mm, rotated rx 180 ry 0 rz -180 deg; joints [1.396, 71.153, -37.474, 2.516, -33.705, -2.094]
  Call Extruder 0.22717
  MoveL (T15926) to (113.64, 121.16, 17.3) mm, rotated rx 180 ry 0 rz -180 deg; joints [1.396, 71.153, -37.474, 2.516, -33.705, -2.094]
  Call Extruder 0.01758
  MoveL (T15927) to (113.07, 121.16, 17.3) mm, rotated rx 180 ry 0 rz -180 deg; joints [3.316, 66.467, -28.663, 5.4, -37.927, -4.264]
  Call Extruder 0.24362
  MoveL (T15928) to (118.71, 115.51, 17.3) mm, rotated rx 180 ry 0 rz -180 deg; joints [3.316, 66.467, -28.663, 5.4, -37.927, -4.264]
  Call Extruder 0.01306
  MoveL (T15929) to (118.52, 115.13, 17.3) mm, rotated rx 180 ry 0 rz -180 deg; joints [2.938, 66.417, -28.57, 4.782, -37.944, -3.774]
  Call Extruder 0.26007
  MoveL (T15930) to (112.49, 121.16, 17.3) mm, rotated rx 180 ry 0 rz -180 deg; joints [2.938, 66.417, -28.57, 4.782, -37.944, -3.774]
  Call Extruder 0.01758
  MoveL (T15931) to (111.91, 121.16, 17.3) mm, rotated rx 180 ry 0 rz -180 deg; joints [3.295, 67.383, -30.384, 5.464, -37.124, -4.361]
  Call Extruder 0.27651
  MoveL (T15932) to (118.32, 114.75, 17.3) mm, rotated rx 180 ry 0 rz -180 deg; joints [3.295, 67.383, -30.384, 5.464, -37.124, -4.361]
  Call Extruder 0.01306
  MoveL (T15933) to (118.13, 114.36, 17.3) mm, rotated rx 180 ry 0 rz -180 deg; joints [3.288, 67.681, -30.944, 5.486, -36.862, -4.394]
  Call Extruder 0.29296
  MoveL (T15934) to (111.34, 121.16, 17.3) mm, rotated rx 180 ry 0 rz -180 deg; joints [3.288, 67.681, -30.944, 5.486, -36.862, -4.394]
  Call Extruder 0.01758
  MoveL (T15935) to (110.76, 121.16, 17.3) mm, rotated rx 180 ry 0 rz -180 deg; joints [1.879, 71.194, -37.551, 3.389, -33.689, -2.821]
  Call Extruder 0.30941
  MoveL (T15936) to (117.93, 113.98, 17.3) mm, rotated rx 180 ry 0 rz -180 deg; joints [1.879, 71.194, -37.551, 3.389, -33.689, -2.821]
  Call Extruder 0.01306
  MoveL (T15937) to (117.74, 113.6, 17.3) mm, rotated rx 180 ry 0 rz -180 deg; joints [1.763, 71.183, -37.531, 3.179, -33.693, -2.646]
  Call Extruder 0.32585
  MoveL (T15938) to (110.18, 121.16, 17.3) mm, rotated rx 180 ry 0 rz -180 deg; joints [1.763, 71.183, -37.531, 3.179, -33.693, -2.646]
  Call Extruder 0.01758
  MoveL (T15939) to (109.61, 121.16, 17.3) mm, rotated rx 180 ry 0 rz -180 deg; joints [1.405, 70.088, -35.47, 2.472, -34.643, -2.034]
  Call Extruder 0.3423
  MoveL (T15940) to (117.54, 113.22, 17.3) mm, rotated rx 180 ry 0 rz -180 deg; joints [1.405, 70.088, -35.47, 2.472, -34.643, -2.034]
  Call Extruder 0.01306
  MoveL (T15941) to (117.35, 112.84, 17.3) mm, rotated rx 180 ry 0 rz -180 deg; joints [1.408, 69.759, -34.852, 2.459, -34.932, -2.017]
  Call Extruder 0.35875
  MoveL (T15942) to (109.03, 121.16, 17.3) mm, rotated rx 180 ry 0 rz -180 deg; joints [1.408, 69.759, -34.852, 2.459, -34.932, -2.017]
  Call Extruder 0.01758
  MoveL (T15943) to (108.45, 121.16, 17.3) mm, rotated rx 180 ry 0 rz -180 deg; joints [1.408, 69.759, -34.852, 2.459, -34.932, -2.017]
  Call Extruder 0.37519
  MoveL (T15944) to (117.15, 112.46, 17.3) mm, rotated rx 180 ry 0 rz -180 deg; joints [2.818, 66.403, -28.543, 4.586, -37.949, -3.619]
  Call Extruder 0.01306
  MoveL (T15945) to (116.96, 112.08, 17.3) mm, rotated rx 180 ry 0 rz -180 deg; joints [2.818, 66.403, -28.543, 4.586, -37.949, -3.619]
  Call Extruder 0.39164
  MoveL (T15946) to (107.88, 121.16, 17.3) mm, rotated rx 180 ry 0 rz -180 deg; joints [2.44, 66.362, -28.466, 3.968, -37.963, -3.13]
  Call Extruder 0.01758
  MoveL (T15947) to (107.3, 121.16, 17.3) mm, rotated rx 180 ry 0 rz -180 deg; joints [2.44, 66.362, -28.466, 3.968, -37.963, -3.13]
  Call Extruder 0.40809
  MoveL (T15948) to (116.76, 111.69, 17.3) mm, rotated rx 180 ry 0 rz -180 deg; joints [3.266, 68.641, -32.749, 5.56, -36.02, -4.502]
  Call Extruder 0.01107
  MoveL (T15949) to (116.6, 111.37, 17.3) mm, rotated rx 180 ry 0 rz -180 deg; joints [3.266, 68.641, -32.749, 5.56, -36.02, -4.502]
  Call Extruder 0.0149
  MoveL (T15950) to (117.09, 111.37, 17.3) mm, rotated rx 180 ry 0 rz -180 deg; joints [3.26, 68.954, -33.338, 5.586, -35.745, -4.538]
  Call Extruder 0.12417
  MoveL (T15951) to (119.96, 108.49, 17.3) mm, rotated rx 180 ry 0 rz -180 deg; joints [3.26, 68.954, -33.338, 5.586, -35.745, -4.538]
  Call Extruder 0.01758
  MoveL (T15952) to (119.96, 107.92, 17.3) mm, rotated rx 180 ry 0 rz -180 deg; joints [3.26, 68.954, -33.338, 5.586, -35.745, -4.538]
  Call Extruder 0.57106
  MoveL (T15953) to (106.73, 121.16, 17.3) mm, rotated rx 180 ry 0 rz -180 deg; joints [2.362, 71.248, -37.652, 4.264, -33.669, -3.551]
  Call Extruder 0.00679
  MoveL (T15954) to (106.5, 121.16, 17.3) mm, rotated rx 180 ry 0 rz -180 deg; joints [2.362, 71.248, -37.652, 4.264, -33.669, -3.551]
  Call Extruder 0.00763
  MoveL (T15955) to (106.33, 120.98, 17.3) mm, rotated rx 180 ry 0 rz -180 deg; joints [2.246, 71.234, -37.625, 4.053, -33.674, -3.374]
  Call Extruder 0.58829
  MoveL (T15956) to (119.96, 107.34, 17.3) mm, rotated rx 180 ry 0 rz -180 deg; joints [2.246, 71.234, -37.625, 4.053, -33.674, -3.374]
  Call Extruder 0.01758
  MoveL (T15957) to (119.96, 106.76, 17.3) mm, rotated rx 180 ry 0 rz -180 deg; joints [2.246, 71.234, -37.625, 4.053, -33.674, -3.374]
  Call Extruder 0.60072
  MoveL (T15958) to (106.04, 120.69, 17.3) mm, rotated rx 180 ry 0 rz -180 deg; joints [1.417, 68.754, -32.963, 2.422, -35.816, -1.964]
  Call Extruder 0.01243
  MoveL (T15959) to (105.75, 120.4, 17.3) mm, rotated rx 180 ry 0 rz -180 deg; joints [1.417, 68.754, -32.963, 2.422, -35.816, -1.964]
  Call Extruder 0.61315
  MoveL (T15960) to (119.96, 106.19, 17.3) mm, rotated rx 180 ry 0 rz -180 deg; joints [1.417, 68.754, -32.963, 2.422, -35.816, -1.964]
  Call Extruder 0.01758
  MoveL (T15961) to (119.96, 105.61, 17.3) mm, rotated rx 180 ry 0 rz -180 deg; joints [1.42, 68.443, -32.377, 2.411, -36.09, -1.949]
  Call Extruder 0.62159
  MoveL (T15962) to (105.55, 120.02, 17.3) mm, rotated rx 180 ry 0 rz -180 deg; joints [1.42, 68.443, -32.377, 2.411, -36.09, -1.949]
  Call Extruder 0.01758
  MoveL (T15963) to (105.55, 119.44, 17.3) mm, rotated rx 180 ry 0 rz -180 deg; joints [2.319, 66.35, -28.443, 3.772, -37.967, -2.975]
  Call Extruder 0.61978
  MoveL (T15964) to (119.92, 105.08, 17.3) mm, rotated rx 180 ry 0 rz -180 deg; joints [2.319, 66.35, -28.443, 3.772, -37.967, -2.975]
  Call Extruder 0.01243
  MoveL (T15965) to (119.63, 104.79, 17.3) mm, rotated rx 180 ry 0 rz -180 deg; joints [2.319, 66.35, -28.443, 3.772, -37.967, -2.975]
  Call Extruder 0.60735
  MoveL (T15966) to (105.55, 118.87, 17.3) mm, rotated rx 180 ry 0 rz -180 deg; joints [1.941, 66.317, -28.381, 3.155, -37.978, -2.488]
  Call Extruder 0.01758
  MoveL (T15967) to (105.55, 118.29, 17.3) mm, rotated rx 180 ry 0 rz -180 deg; joints [1.941, 66.317, -28.381, 3.155, -37.978, -2.488]
  Call Extruder 0.59492
  MoveL (T15968) to (119.35, 104.5, 17.3) mm, rotated rx 180 ry 0 rz -180 deg; joints [1.941, 66.317, -28.381, 3.155, -37.978, -2.488]
  Call Extruder 0.01243
  MoveL (T15969) to (119.06, 104.21, 17.3) mm, rotated rx 180 ry 0 rz -180 deg; joints [1.941, 66.317, -28.381, 3.155, -37.978, -2.488]
  Call Extruder 0.58249
  MoveL (T15970) to (105.55, 117.72, 17.3) mm, rotated rx 180 ry 0 rz -180 deg; joints [3.239, 69.966, -35.241, 5.673, -34.856, -4.66]
  Call Extruder 0.01758
  MoveL (T15971) to (105.55, 117.14, 17.3) mm, rotated rx 180 ry 0 rz -180 deg; joints [3.239, 69.966, -35.241, 5.673, -34.856, -4.66]
  Call Extruder 0.57006
  MoveL (T15972) to (118.77, 103.92, 17.3) mm, rotated rx 180 ry 0 rz -180 deg; joints [3.239, 69.966, -35.241, 5.673, -34.856, -4.66]
  Call Extruder 0.00343
  MoveL (T15973) to (118.69, 103.84, 17.3) mm, rotated rx 180 ry 0 rz -180 deg; joints [3.232, 70.297, -35.864, 5.703, -34.566, -4.701]
  Call Extruder 0.01274
  MoveL (T15974) to (118.27, 103.84, 17.3) mm, rotated rx 180 ry 0 rz -180 deg; joints [3.232, 70.297, -35.864, 5.703, -34.566, -4.701]
  Call Extruder 0.54862
  MoveL (T15975) to (105.55, 116.56, 17.3) mm, rotated rx 180 ry 0 rz -180 deg; joints [3.232, 70.297, -35.864, 5.703, -34.566, -4.701]
  Call Extruder 0.01758
  MoveL (T15976) to (105.55, 115.99, 17.3) mm, rotated rx 180 ry 0 rz -180 deg; joints [2.845, 71.313, -37.775, 5.14, -33.644, -4.283]
  Call Extruder 0.0956
  MoveL (T15977) to (107.77, 113.77, 17.3) mm, rotated rx 180 ry 0 rz -180 deg; joints [2.845, 71.313, -37.775, 5.14, -33.644, -4.283]
  Set speed (150.0 mm/s)
  MoveL (T15978) to (108.15, 113.39, 17.3) mm, rotated rx 180 ry 0 rz -180 deg; joints [2.845, 71.313, -37.775, 5.14, -33.644, -4.283]
  Set speed (40.0 mm/s)
  MoveL (T15979) to (108.15, 113.39, 17.3) mm, rotated rx 180 ry 0 rz -180 deg; joints [2.729, 71.296, -37.743, 4.929, -33.651, -4.106]
  Call Extruder 0.41176
  MoveL (T15980) to (117.7, 103.84, 17.3) mm, rotated rx 180 ry 0 rz -180 deg; joints [2.729, 71.296, -37.743, 4.929, -33.651, -4.106]
  Call Extruder 0.01758
  MoveL (T15981) to (117.12, 103.84, 17.3) mm, rotated rx 180 ry 0 rz -180 deg; joints [1.429, 67.489, -30.584, 2.379, -36.929, -1.902]
  Call Extruder 0.38942
  MoveL (T15982) to (108.09, 112.87, 17.3) mm, rotated rx 180 ry 0 rz -180 deg; joints [1.429, 67.489, -30.584, 2.379, -36.929, -1.902]
  Call Extruder 0.01307
  MoveL (T15983) to (107.9, 112.49, 17.3) mm, rotated rx 180 ry 0 rz -180 deg; joints [1.429, 67.489, -30.584, 2.379, -36.929, -1.902]
  Call Extruder 0.37296
  MoveL (T15984) to (116.54, 103.84, 17.3) mm, rotated rx 180 ry 0 rz -180 deg; joints [1.432, 67.193, -30.027, 2.37, -37.189, -1.888]
  Call Extruder 0.01758
  MoveL (T15985) to (115.97, 103.84, 17.3) mm, rotated rx 180 ry 0 rz -180 deg; joints [1.432, 67.193, -30.027, 2.37, -37.189, -1.888]
  Call Extruder 0.35649
  MoveL (T15986) to (107.7, 112.11, 17.3) mm, rotated rx 180 ry 0 rz -180 deg; joints [1.432, 67.193, -30.027, 2.37, -37.189, -1.888]
  Call Extruder 0.01307
  MoveL (T15987) to (107.51, 111.73, 17.3) mm, rotated rx 180 ry 0 rz -180 deg; joints [1.821, 66.307, -28.363, 2.959, -37.981, -2.333]
  Call Extruder 0.34003
  MoveL (T15988) to (115.39, 103.84, 17.3) mm, rotated rx 180 ry 0 rz -180 deg; joints [1.821, 66.307, -28.363, 2.959, -37.981, -2.333]
  Call Extruder 0.01758
  MoveL (T15989) to (114.81, 103.84, 17.3) mm, rotated rx 180 ry 0 rz -180 deg; joints [1.821, 66.307, -28.363, 2.959, -37.981, -2.333]
  Call Extruder 0.32357
  MoveL (T15990) to (107.31, 111.35, 17.3) mm, rotated rx 180 ry 0 rz -180 deg; joints [1.442, 66.282, -28.315, 2.343, -37.99, -1.847]
  Call Extruder 0.01307
  MoveL (T15991) to (107.12, 110.96, 17.3) mm, rotated rx 180 ry 0 rz -180 deg; joints [1.442, 66.282, -28.315, 2.343, -37.99, -1.847]
  Call Extruder 0.3071
  MoveL (T15992) to (114.24, 103.84, 17.3) mm, rotated rx 180 ry 0 rz -180 deg; joints [3.211, 71.372, -37.885, 5.806, -33.623, -4.84]
  Call Extruder 0.01758
  MoveL (T15993) to (113.66, 103.84, 17.3) mm, rotated rx 180 ry 0 rz -180 deg; joints [3.211, 71.372, -37.885, 5.806, -33.623, -4.84]
  Call Extruder 0.29064
  MoveL (T15994) to (106.92, 110.58, 17.3) mm, rotated rx 180 ry 0 rz -180 deg; joints [3.226, 70.615, -36.462, 5.733, -34.287, -4.741]
  Call Extruder 0.01307
  MoveL (T15995) to (106.73, 110.2, 17.3) mm, rotated rx 180 ry 0 rz -180 deg; joints [3.226, 70.615, -36.462, 5.733, -34.287, -4.741]
  Call Extruder 0.27417
  MoveL (T15996) to (113.08, 103.84, 17.3) mm, rotated rx 180 ry 0 rz -180 deg; joints [3.226, 70.615, -36.462, 5.733, -34.287, -4.741]
  Call Extruder 0.01758
  MoveL (T15997) to (112.51, 103.84, 17.3) mm, rotated rx 180 ry 0 rz -180 deg; joints [3.226, 70.615, -36.462, 5.733, -34.287, -4.741]
  Call Extruder 0.25771
  MoveL (T15998) to (106.53, 109.82, 17.3) mm, rotated rx 180 ry 0 rz -180 deg; joints [3.226, 70.615, -36.462, 5.733, -34.287, -4.741]
  Call Extruder 0.01307
  MoveL (T15999) to (106.34, 109.44, 17.3) mm, rotated rx 180 ry 0 rz -180 deg; joints [3.226, 70.615, -36.462, 5.733, -34.287, -4.741]
  Call Extruder 0.24124
  MoveL (T16000) to (111.93, 103.84, 17.3) mm, rotated rx 180 ry 0 rz -180 deg; joints [3.226, 70.615, -36.462, 5.733, -34.287, -4.741]
  Call Extruder 0.01758
  MoveL (T16001) to (111.36, 103.84, 17.3) mm, rotated rx 180 ry 0 rz -180 deg; joints [3.219, 70.942, -37.078, 5.764, -33.999, -4.784]
  Call Extruder 0.22478
  MoveL (T16002) to (106.14, 109.06, 17.3) mm, rotated rx 180 ry 0 rz -180 deg; joints [3.219, 70.942, -37.078, 5.764, -33.999, -4.784]
  Call Extruder 0.01307
  MoveL (T16003) to (105.95, 108.67, 17.3) mm, rotated rx 180 ry 0 rz -180 deg; joints [3.219, 70.942, -37.078, 5.764, -33.999, -4.784]
  Call Extruder 0.20831
  MoveL (T16004) to (110.78, 103.84, 17.3) mm, rotated rx 180 ry 0 rz -180 deg; joints [3.219, 70.708, -37.033, 5.792, -33.811, -4.818]
  Call Extruder 0.01758
  MoveL (T16005) to (110.2, 103.84, 17.3) mm, rotated rx 180 ry 0 rz -180 deg; joints [3.219, 70.708, -37.033, 5.792, -33.811, -4.818]
  Call Extruder 0.19185
  MoveL (T16006) to (105.75, 108.29, 17.3) mm, rotated rx 180 ry 0 rz -180 deg; joints [1.407, 66.17, -28.512, 2.303, -37.68, -1.823]
  Call Extruder 0.00693
  MoveL (T16007) to (105.65, 108.09, 17.3) mm, rotated rx 180 ry 0 rz -180 deg; joints [1.407, 66.383, -28.547, 2.293, -37.859, -1.811]
  Call Extruder 0.00686
  MoveL (T16008) to (105.6, 107.87, 17.3) mm, rotated rx 180 ry 0 rz -180 deg; joints [1.407, 66.383, -28.547, 2.293, -37.859, -1.811]
  Call Extruder 0.17364
  MoveL (T16009) to (109.63, 103.84, 17.3) mm, rotated rx 180 ry 0 rz -180 deg; joints [1.407, 66.383, -28.547, 2.293, -37.859, -1.811]
  Call Extruder 0.01758
  MoveL (T16010) to (109.05, 103.84, 17.3) mm, rotated rx 180 ry 0 rz -180 deg; joints [1.407, 66.383, -28.547, 2.293, -37.859, -1.811]
  Call Extruder 0.15359
  MoveL (T16011) to (105.49, 107.41, 17.3) mm, rotated rx 180 ry 0 rz -180 deg; joints [1.407, 66.383, -28.547, 2.293, -37.859, -1.811]
  Call Extruder 0.00278
  MoveL (T16012) to (105.47, 107.32, 17.3) mm, rotated rx 180 ry 0 rz -180 deg; joints [1.407, 66.383, -28.547, 2.293, -37.859, -1.811]
  Call Extruder 0.01427
  MoveL (T16013) to (105.47, 106.85, 17.3) mm, rotated rx 180 ry 0 rz -180 deg; joints [1.363, 71.223, -37.644, 2.464, -33.603, -2.052]
  Call Extruder 0.12957
  MoveL (T16014) to (108.47, 103.84, 17.3) mm, rotated rx 180 ry 0 rz -180 deg; joints [1.363, 71.223, -37.644, 2.464, -33.603, -2.052]
  Call Extruder 0.01758
  MoveL (T16015) to (107.9, 103.84, 17.3) mm, rotated rx 180 ry 0 rz -180 deg; joints [3.241, 71.45, -38.071, 5.877, -33.517, -4.905]
  Call Extruder 0.1047
  MoveL (T16016) to (105.47, 106.27, 17.3) mm, rotated rx 180 ry 0 rz -180 deg; joints [3.351, 66.369, -28.52, 5.451, -37.975, -4.302]
  Call Extruder 0.01758
  MoveL (T16017) to (105.47, 105.69, 17.3) mm, rotated rx 180 ry 0 rz -180 deg; joints [3.351, 66.369, -28.52, 5.451, -37.975, -4.302]
  Call Extruder 0.07984
  MoveL (T16018) to (107.32, 103.84, 17.3) mm, rotated rx 180 ry 0 rz -180 deg; joints [1.409, 66.178, -28.161, 2.288, -38.039, -1.802]
  Call Extruder 0.01758
  MoveL (T16019) to (106.75, 103.84, 17.3) mm, rotated rx 180 ry 0 rz -180 deg; joints [1.407, 66.368, -28.518, 2.293, -37.872, -1.81]
  Call Extruder 0.06288
  MoveL (T16020) to (105.29, 105.3, 17.3) mm, rotated rx 180 ry 0 rz -180 deg; joints [1.407, 66.368, -28.518, 2.293, -37.872, -1.81]
  Set speed (45.0 mm/s)
  Call Extruder -1.6
  MoveL (T16021) to (105.29, 105.3, 17.3) mm, rotated rx 180 ry 0 rz -180 deg; joints [1.365, 66.174, -28.153, 2.216, -38.042, -1.746]
  Set speed (120.0 mm/s)
  MoveL (T16022) to (105.29, 105.3, 17.3) mm, rotated rx 180 ry 0 rz -180 deg; joints [1.365, 66.174, -28.153, 2.216, -38.042, -1.746]
  Call Extruder -0.38
  MoveL (T16023) to (106.04, 104.55, 17.3) mm, rotated rx 180 ry 0 rz -180 deg; joints [1.365, 66.174, -28.153, 2.216, -38.042, -1.746]
  Set speed (45.0 mm/s)
  Call Extruder -0.02
  MoveL (T16024) to (106.04, 104.55, 17.3) mm, rotated rx 180 ry 0 rz -180 deg; joints [1.319, 71.348, -37.879, 2.392, -33.491, -1.995]
  Set speed (150.0 mm/s)
  MoveL (T16025) to (106.04, 104.55, 19.3) mm, rotated rx 180 ry 0 rz -180 deg; joints [1.319, 71.348, -37.879, 2.392, -33.491, -1.995]
  MoveL (T16026) to (104.34, 103.54, 19.3) mm, rotated rx 180 ry 0 rz -180 deg; joints [1.319, 71.348, -37.879, 2.392, -33.491, -1.995]
  MoveL (T16027) to (104.34, 103.54, 17.5) mm, rotated rx 180 ry 0 rz -180 deg; joints [3.282, 71.586, -38.328, 5.969, -33.401, -4.988]
  Set speed (40.0 mm/s)
  Call Extruder 2.0
  MoveL (T16028) to (104.34, 103.54, 17.5) mm, rotated rx 180 ry 0 rz -180 deg; joints [3.398, 66.271, -28.335, 5.516, -38.065, -4.348]
  Call Extruder 0.52159
  MoveL (T16029) to (121.46, 103.54, 17.5) mm, rotated rx 180 ry 0 rz -180 deg; joints [3.398, 66.271, -28.335, 5.516, -38.065, -4.348]
  Call Extruder 0.54596
  MoveL (T16030) to (121.46, 121.46, 17.5) mm, rotated rx 180 ry 0 rz -180 deg; joints [3.398, 66.271, -28.335, 5.516, -38.065, -4.348]
  Call Extruder 0.54596
  MoveL (T16031) to (103.54, 121.46, 17.5) mm, rotated rx 180 ry 0 rz -180 deg; joints [1.366, 66.072, -27.961, 2.213, -38.131, -1.741]
  Call Extruder 0.54596
  MoveL (T16032) to (103.54, 103.54, 17.5) mm, rotated rx 180 ry 0 rz -180 deg; joints [1.366, 66.072, -27.961, 2.213, -38.131, -1.741]
  Call Extruder 0.02254
  MoveL (T16033) to (104.28, 103.54, 17.5) mm, rotated rx 180 ry 0 rz -180 deg; joints [1.366, 66.072, -27.961, 2.213, -38.131, -1.741]
  Set speed (150.0 mm/s)
  MoveL (T16034) to (103.53, 103.13, 17.5) mm, rotated rx 180 ry 0 rz -180 deg; joints [1.365, 66.158, -28.124, 2.215, -38.055, -1.745]
  Set speed (40.0 mm/s)
  MoveL (T16035) to (103.53, 103.13, 17.5) mm, rotated rx 180 ry 0 rz -180 deg; joints [1.332, 65.966, -27.763, 2.154, -38.223, -1.692]
  Call Extruder 0.55858
  MoveL (T16036) to (121.87, 103.13, 17.5) mm, rotated rx 180 ry 0 rz -180 deg; joints [1.332, 65.966, -27.763, 2.154, -38.223, -1.692]
  Call Extruder 0.57077
  MoveL (T16037) to (121.87, 121.87, 17.5) mm, rotated rx 180 ry 0 rz -180 deg; joints [1.332, 65.966, -27.763, 2.154, -38.223, -1.692]
  Call Extruder 0.57077
  MoveL (T16038) to (103.13, 121.87, 17.5) mm, rotated rx 180 ry 0 rz -180 deg; joints [1.332, 65.966, -27.763, 2.154, -38.223, -1.692]
  Call Extruder 0.57077
  MoveL (T16039) to (103.13, 103.13, 17.5) mm, rotated rx 180 ry 0 rz -180 deg; joints [1.332, 65.966, -27.763, 2.154, -38.223, -1.692]
  Call Extruder 0.01036
  MoveL (T16040) to (103.47, 103.13, 17.5) mm, rotated rx 180 ry 0 rz -180 deg; joints [1.332, 65.966, -27.763, 2.154, -38.223, -1.692]
  Set speed (150.0 mm/s)
  MoveL (T16041) to (102.72, 102.81, 17.5) mm, rotated rx 180 ry 0 rz -180 deg; joints [1.332, 65.966, -27.763, 2.154, -38.223, -1.692]
  Set speed (25.0 mm/s)
  MoveL (T16042) to (102.72, 102.81, 17.5) mm, rotated rx 180 ry 0 rz -180 deg; joints [1.332, 65.966, -27.763, 2.154, -38.223, -1.692]
  Call Extruder 0.00259
  MoveL (T16043) to (102.72, 102.72, 17.5) mm, rotated rx 180 ry 0 rz -180 deg; joints [1.323, 65.966, -27.762, 2.139, -38.223, -1.681]
  Call Extruder 0.59557
  MoveL (T16044) to (122.28, 102.72, 17.5) mm, rotated rx 180 ry 0 rz -180 deg; joints [1.323, 65.966, -27.762, 2.139, -38.223, -1.681]
  Call Extruder 0.59557
  MoveL (T16045) to (122.28, 122.28, 17.5) mm, rotated rx 180 ry 0 rz -180 deg; joints [1.323, 65.966, -27.762, 2.139, -38.223, -1.681]
  Call Extruder 0.59557
  MoveL (T16046) to (102.72, 122.28, 17.5) mm, rotated rx 180 ry 0 rz -180 deg; joints [1.323, 65.966, -27.762, 2.139, -38.223, -1.681]
  Call Extruder 0.59115
  MoveL (T16047) to (102.72, 102.87, 17.5) mm, rotated rx 180 ry 0 rz -180 deg; joints [1.276, 71.474, -38.116, 2.319, -33.379, -1.937]
  Set speed (150.0 mm/s)
  MoveL (T16048) to (102.78, 102.75, 17.5) mm, rotated rx 180 ry 0 rz -180 deg; joints [1.276, 71.474, -38.116, 2.319, -33.379, -1.937]
  Set speed (45.0 mm/s)
  Call Extruder -1.6
  MoveL (T16049) to (102.78, 102.75, 17.5) mm, rotated rx 180 ry 0 rz -180 deg; joints [3.322, 71.724, -38.587, 6.06, -33.284, -5.072]
  Set speed (120.0 mm/s)
  MoveL (T16050) to (102.78, 102.75, 17.5) mm, rotated rx 180 ry 0 rz -180 deg; joints [3.322, 71.724, -38.587, 6.06, -33.284, -5.072]
  Call Extruder -0.05166
  MoveL (T16051) to (102.72, 102.72, 17.5) mm, rotated rx 180 ry 0 rz -180 deg; joints [3.322, 71.724, -38.587, 6.06, -33.284, -5.072]
  Call Extruder -0.32834
  MoveL (T16052) to (103.65, 102.72, 17.5) mm, rotated rx 180 ry 0 rz -180 deg; joints [3.445, 66.173, -28.151, 5.581, -38.154, -4.394]
  Set speed (45.0 mm/s)
  Call Extruder -0.02
  MoveL (T16053) to (103.65, 102.72, 17.5) mm, rotated rx 180 ry 0 rz -180 deg; joints [3.445, 66.173, -28.151, 5.581, -38.154, -4.394]
  Set speed (150.0 mm/s)
  MoveL (T16054) to (103.65, 102.72, 19.5) mm, rotated rx 180 ry 0 rz -180 deg; joints [3.445, 66.173, -28.151, 5.581, -38.154, -4.394]
  MoveL (T16055) to (106.08, 103.93, 19.5) mm, rotated rx 180 ry 0 rz -180 deg; joints [1.339, 65.967, -27.764, 2.164, -38.223, -1.701]
  MoveL (T16056) to (106.08, 103.93, 17.5) mm, rotated rx 180 ry 0 rz -180 deg; joints [1.339, 65.967, -27.764, 2.164, -38.223, -1.701]
  Set speed (40.0 mm/s)
  Call Extruder 2.0
  MoveL (T16057) to (106.08, 103.93, 17.5) mm, rotated rx 180 ry 0 rz -180 deg; joints [1.339, 65.967, -27.764, 2.164, -38.223, -1.701]
  Set speed (50.0 mm/s)
  MoveL (T16058) to (106.08, 103.93, 17.5) mm, rotated rx 180 ry 0 rz -180 deg; joints [1.326, 65.981, -27.791, 2.144, -38.21, -1.685]
  Call Extruder 0.00361
  MoveL (T16059) to (106.17, 103.84, 17.5) mm, rotated rx 180 ry 0 rz -180 deg; joints [1.326, 65.981, -27.791, 2.144, -38.21, -1.685]
  Call Extruder 0.0708
  MoveL (T16060) to (103.84, 103.84, 17.5) mm, rotated rx 180 ry 0 rz -180 deg; joints [1.326, 65.981, -27.791, 2.144, -38.21, -1.685]
  Call Extruder 0.05255
  MoveL (T16061) to (105.06, 105.06, 17.5) mm, rotated rx 180 ry 0 rz -180 deg; joints [1.326, 65.981, -27.791, 2.144, -38.21, -1.685]
  Call Extruder 0.03217
  MoveL (T16062) to (105.06, 106.12, 17.5) mm, rotated rx 180 ry 0 rz -180 deg; joints [1.326, 65.981, -27.791, 2.144, -38.21, -1.685]
  Call Extruder 0.0525
  MoveL (T16063) to (103.84, 107.34, 17.5) mm, rotated rx 180 ry 0 rz -180 deg; joints [1.326, 65.981, -27.791, 2.144, -38.21, -1.685]
  Call Extruder 0.03385
  MoveL (T16064) to (103.84, 108.45, 17.5) mm, rotated rx 180 ry 0 rz -180 deg; joints [1.326, 65.981, -27.791, 2.144, -38.21, -1.685]
  Call Extruder 0.13495
  MoveL (T16065) to (106.98, 111.58, 17.5) mm, rotated rx 180 ry 0 rz -180 deg; joints [1.326, 65.981, -27.791, 2.144, -38.21, -1.685]
  Call Extruder 0.04156
  MoveL (T16066) to (107.6, 112.8, 17.5) mm, rotated rx 180 ry 0 rz -180 deg; joints [1.326, 65.981, -27.791, 2.144, -38.21, -1.685]
  Call Extruder 0.16166
  MoveL (T16067) to (103.84, 116.55, 17.5) mm, rotated rx 180 ry 0 rz -180 deg; joints [1.326, 65.981, -27.791, 2.144, -38.21, -1.685]
  Call Extruder 0.03385
  MoveL (T16068) to (103.84, 117.66, 17.5) mm, rotated rx 180 ry 0 rz -180 deg; joints [1.326, 65.981, -27.791, 2.144, -38.21, -1.685]
  Call Extruder 0.05612
  MoveL (T16069) to (105.15, 118.96, 17.5) mm, rotated rx 180 ry 0 rz -180 deg; joints [1.326, 65.981, -27.791, 2.144, -38.21, -1.685]
  Call Extruder 0.02709
  MoveL (T16070) to (105.15, 119.85, 17.5) mm, rotated rx 180 ry 0 rz -180 deg; joints [1.326, 65.981, -27.791, 2.144, -38.21, -1.685]
  Call Extruder 0.05612
  MoveL (T16071) to (103.84, 121.16, 17.5) mm, rotated rx 180 ry 0 rz -180 deg; joints [1.323, 65.966, -27.762, 2.139, -38.223, -1.681]
  Call Extruder 0.06345
  MoveL (T16072) to (105.93, 121.16, 17.5) mm, rotated rx 180 ry 0 rz -180 deg; joints [1.323, 65.966, -27.762, 2.139, -38.223, -1.681]
  Call Extruder 0.01096
  MoveL (T16073) to (105.67, 120.9, 17.5) mm, rotated rx 180 ry 0 rz -180 deg; joints [1.323, 65.966, -27.762, 2.139, -38.223, -1.681]
  Set speed (45.0 mm/s)
  Call Extruder -1.6
  MoveL (T16074) to (105.67, 120.9, 17.5) mm, rotated rx 180 ry 0 rz -180 deg; joints [1.321, 66.201, -28.203, 2.145, -38.017, -1.69]
  Set speed (120.0 mm/s)
  MoveL (T16075) to (105.67, 120.9, 17.5) mm, rotated rx 180 ry 0 rz -180 deg; joints [1.321, 66.201, -28.203, 2.145, -38.017, -1.69]
  Call Extruder -0.12811
  MoveL (T16076) to (105.93, 121.16, 17.5) mm, rotated rx 180 ry 0 rz -180 deg; joints [1.321, 66.201, -28.203, 2.145, -38.017, -1.69]
  Call Extruder -0.25189
  MoveL (T16077) to (105.22, 121.16, 17.5) mm, rotated rx 180 ry 0 rz -180 deg; joints [1.321, 66.201, -28.203, 2.145, -38.017, -1.69]
  Set speed (45.0 mm/s)
  Call Extruder -0.02
  MoveL (T16078) to (105.22, 121.16, 17.5) mm, rotated rx 180 ry 0 rz -180 deg; joints [1.321, 66.201, -28.203, 2.145, -38.017, -1.69]
  Set speed (150.0 mm/s)
  MoveL (T16079) to (105.22, 121.16, 19.5) mm, rotated rx 180 ry 0 rz -180 deg; joints [1.321, 66.201, -28.203, 2.145, -38.017, -1.69]
  MoveL (T16080) to (105.15, 117.23, 19.5) mm, rotated rx 180 ry 0 rz -180 deg; joints [1.321, 66.201, -28.203, 2.145, -38.017, -1.69]
  MoveL (T16081) to (105.15, 117.23, 17.5) mm, rotated rx 180 ry 0 rz -180 deg; joints [1.321, 66.201, -28.203, 2.145, -38.017, -1.69]
  Set speed (40.0 mm/s)
  Call Extruder 2.0
  MoveL (T16082) to (105.15, 117.23, 17.5) mm, rotated rx 180 ry 0 rz -180 deg; joints [1.321, 66.201, -28.203, 2.145, -38.017, -1.69]
  Set speed (50.0 mm/s)
  MoveL (T16083) to (105.15, 117.23, 17.5) mm, rotated rx 180 ry 0 rz -180 deg; joints [1.321, 65.963, -28.166, 2.155, -37.817, -1.702]
  Call Extruder 0.04143
  MoveL (T16084) to (105.15, 115.87, 17.5) mm, rotated rx 180 ry 0 rz -180 deg; joints [1.402, 70.379, -36.059, 2.486, -34.346, -2.053]
  Call Extruder 0.00661
  MoveL (T16085) to (105.23, 115.67, 17.5) mm, rotated rx 180 ry 0 rz -180 deg; joints [1.402, 70.379, -36.059, 2.486, -34.346, -2.053]
  Call Extruder 0.02637
  MoveL (T16086) to (105.84, 115.05, 17.5) mm, rotated rx 180 ry 0 rz -180 deg; joints [1.402, 70.379, -36.059, 2.486, -34.346, -2.053]
  Call Extruder 0.08606
  MoveL (T16087) to (103.84, 113.06, 17.5) mm, rotated rx 180 ry 0 rz -180 deg; joints [1.402, 70.379, -36.059, 2.486, -34.346, -2.053]
  Call Extruder 0.03385
  MoveL (T16088) to (103.84, 111.94, 17.5) mm, rotated rx 180 ry 0 rz -180 deg; joints [1.402, 70.379, -36.059, 2.486, -34.346, -2.053]
  Call Extruder 0.09463
  MoveL (T16089) to (106.04, 109.75, 17.5) mm, rotated rx 180 ry 0 rz -180 deg; joints [1.402, 70.379, -36.059, 2.486, -34.346, -2.053]
  Call Extruder 0.05062
  MoveL (T16090) to (105.29, 108.27, 17.5) mm, rotated rx 180 ry 0 rz -180 deg; joints [1.402, 70.379, -36.059, 2.486, -34.346, -2.053]
  Call Extruder 0.02377
  MoveL (T16091) to (105.1, 107.51, 17.5) mm, rotated rx 180 ry 0 rz -180 deg; joints [1.402, 70.379, -36.059, 2.486, -34.346, -2.053]
  Set speed (45.0 mm/s)
  Call Extruder -1.6
  MoveL (T16092) to (105.1, 107.51, 17.5) mm, rotated rx 180 ry 0 rz -180 deg; joints [1.402, 70.379, -36.059, 2.486, -34.346, -2.053]
  Set speed (120.0 mm/s)
  MoveL (T16093) to (105.1, 107.51, 17.5) mm, rotated rx 180 ry 0 rz -180 deg; joints [1.396, 71.13, -37.469, 2.517, -33.686, -2.095]
  Call Extruder -0.278
  MoveL (T16094) to (105.29, 108.27, 17.5) mm, rotated rx 180 ry 0 rz -180 deg; joints [1.396, 71.13, -37.469, 2.517, -33.686, -2.095]
  Call Extruder -0.102
  MoveL (T16095) to (105.42, 108.52, 17.5) mm, rotated rx 180 ry 0 rz -180 deg; joints [1.396, 71.13, -37.469, 2.517, -33.686, -2.095]
  Set speed (45.0 mm/s)
  Call Extruder -0.02
  MoveL (T16096) to (105.42, 108.52, 17.5) mm, rotated rx 180 ry 0 rz -180 deg; joints [3.316, 66.443, -28.659, 5.403, -37.908, -4.267]
  Set speed (150.0 mm/s)
  MoveL (T16097) to (105.42, 108.52, 19.5) mm, rotated rx 180 ry 0 rz -180 deg; joints [3.316, 66.443, -28.659, 5.403, -37.908, -4.267]
  MoveL (T16098) to (118.51, 103.66, 19.5) mm, rotated rx 180 ry 0 rz -180 deg; joints [3.316, 66.443, -28.659, 5.403, -37.908, -4.267]
  MoveL (T16099) to (118.51, 103.66, 17.5) mm, rotated rx 180 ry 0 rz -180 deg; joints [3.316, 66.443, -28.659, 5.403, -37.908, -4.267]
  Set speed (40.0 mm/s)
  Call Extruder 2.0
  MoveL (T16100) to (118.51, 103.66, 17.5) mm, rotated rx 180 ry 0 rz -180 deg; joints [2.938, 66.394, -28.566, 4.784, -37.924, -3.777]
  Call Extruder 0.06226
  MoveL (T16101) to (119.94, 105.1, 17.5) mm, rotated rx 180 ry 0 rz -180 deg; joints [2.938, 66.394, -28.566, 4.784, -37.924, -3.777]
  Call Extruder 0.00161
  MoveL (T16102) to (119.96, 105.15, 17.5) mm, rotated rx 180 ry 0 rz -180 deg; joints [2.938, 66.394, -28.566, 4.784, -37.924, -3.777]
  Call Extruder 0.01683
  MoveL (T16103) to (119.96, 105.7, 17.5) mm, rotated rx 180 ry 0 rz -180 deg; joints [3.295, 67.359, -30.38, 5.466, -37.104, -4.364]
  Call Extruder 0.08024
  MoveL (T16104) to (118.11, 103.84, 17.5) mm, rotated rx 180 ry 0 rz -180 deg; joints [3.295, 67.359, -30.38, 5.466, -37.104, -4.364]
  Call Extruder 0.0177
  MoveL (T16105) to (117.53, 103.84, 17.5) mm, rotated rx 180 ry 0 rz -180 deg; joints [3.295, 67.359, -30.38, 5.466, -37.104, -4.364]
  Call Extruder 0.10527
  MoveL (T16106) to (119.96, 106.28, 17.5) mm, rotated rx 180 ry 0 rz -180 deg; joints [3.295, 67.359, -30.38, 5.466, -37.104, -4.364]
  Call Extruder 0.0177
  MoveL (T16107) to (119.96, 106.86, 17.5) mm, rotated rx 180 ry 0 rz -180 deg; joints [3.288, 67.657, -30.94, 5.488, -36.843, -4.397]
  Call Extruder 0.1303
  MoveL (T16108) to (116.95, 103.84, 17.5) mm, rotated rx 180 ry 0 rz -180 deg; joints [3.288, 67.657, -30.94, 5.488, -36.843, -4.397]
  Call Extruder 0.0177
  MoveL (T16109) to (116.38, 103.84, 17.5) mm, rotated rx 180 ry 0 rz -180 deg; joints [3.288, 67.657, -30.94, 5.488, -36.843, -4.397]
  Call Extruder 0.15533
  MoveL (T16110) to (119.96, 107.43, 17.5) mm, rotated rx 180 ry 0 rz -180 deg; joints [3.288, 67.657, -30.94, 5.488, -36.843, -4.397]
  Call Extruder 0.0177
  MoveL (T16111) to (119.96, 108.01, 17.5) mm, rotated rx 180 ry 0 rz -180 deg; joints [1.879, 71.171, -37.547, 3.391, -33.67, -2.823]
  Call Extruder 0.18036
  MoveL (T16112) to (115.8, 103.84, 17.5) mm, rotated rx 180 ry 0 rz -180 deg; joints [1.879, 71.171, -37.547, 3.391, -33.67, -2.823]
  Call Extruder 0.0177
  MoveL (T16113) to (115.22, 103.84, 17.5) mm, rotated rx 180 ry 0 rz -180 deg; joints [1.879, 71.171, -37.547, 3.391, -33.67, -2.823]
  Call Extruder 0.20539
  MoveL (T16114) to (119.96, 108.59, 17.5) mm, rotated rx 180 ry 0 rz -180 deg; joints [1.763, 71.16, -37.526, 3.18, -33.675, -2.647]
  Call Extruder 0.0177
  MoveL (T16115) to (119.96, 109.17, 17.5) mm, rotated rx 180 ry 0 rz -180 deg; joints [1.763, 71.16, -37.526, 3.18, -33.675, -2.647]
  Call Extruder 0.23042
  MoveL (T16116) to (114.64, 103.84, 17.5) mm, rotated rx 180 ry 0 rz -180 deg; joints [1.763, 71.16, -37.526, 3.18, -33.675, -2.647]
  Call Extruder 0.0177
  MoveL (T16117) to (114.06, 103.84, 17.5) mm, rotated rx 180 ry 0 rz -180 deg; joints [1.763, 71.16, -37.526, 3.18, -33.675, -2.647]
  Call Extruder 0.24813
  MoveL (T16118) to (119.8, 109.58, 17.5) mm, rotated rx 180 ry 0 rz -180 deg; joints [1.763, 71.16, -37.526, 3.18, -33.675, -2.647]
  Call Extruder 0.01252
  MoveL (T16119) to (119.51, 109.87, 17.5) mm, rotated rx 180 ry 0 rz -180 deg; joints [1.405, 70.064, -35.465, 2.473, -34.624, -2.036]
  Call Extruder 0.26064
  MoveL (T16120) to (113.48, 103.84, 17.5) mm, rotated rx 180 ry 0 rz -180 deg; joints [1.408, 69.735, -34.848, 2.46, -34.913, -2.018]
  Call Extruder 0.0177
  MoveL (T16121) to (112.91, 103.84, 17.5) mm, rotated rx 180 ry 0 rz -180 deg; joints [1.408, 69.735, -34.848, 2.46, -34.913, -2.018]
  Call Extruder 0.27316
  MoveL (T16122) to (119.22, 110.16, 17.5) mm, rotated rx 180 ry 0 rz -180 deg; joints [2.818, 66.379, -28.539, 4.588, -37.929, -3.621]
  Call Extruder 0.01252
  MoveL (T16123) to (118.93, 110.44, 17.5) mm, rotated rx 180 ry 0 rz -180 deg; joints [2.818, 66.379, -28.539, 4.588, -37.929, -3.621]
  Call Extruder 0.28567
  MoveL (T16124) to (112.33, 103.84, 17.5) mm, rotated rx 180 ry 0 rz -180 deg; joints [2.44, 66.338, -28.462, 3.97, -37.943, -3.133]
  Call Extruder 0.0177
  MoveL (T16125) to (111.75, 103.84, 17.5) mm, rotated rx 180 ry 0 rz -180 deg; joints [2.44, 66.338, -28.462, 3.97, -37.943, -3.133]
  Call Extruder 0.29819
  MoveL (T16126) to (118.64, 110.73, 17.5) mm, rotated rx 180 ry 0 rz -180 deg; joints [3.266, 68.617, -32.745, 5.563, -36.001, -4.505]
  Call Extruder 0.01252
  MoveL (T16127) to (118.35, 111.02, 17.5) mm, rotated rx 180 ry 0 rz -180 deg; joints [3.266, 68.617, -32.745, 5.563, -36.001, -4.505]
  Call Extruder 0.3107
  MoveL (T16128) to (111.17, 103.84, 17.5) mm, rotated rx 180 ry 0 rz -180 deg; joints [3.26, 68.93, -33.334, 5.588, -35.726, -4.542]
  Call Extruder 0.0177
  MoveL (T16129) to (110.59, 103.84, 17.5) mm, rotated rx 180 ry 0 rz -180 deg; joints [3.26, 68.93, -33.334, 5.588, -35.726, -4.542]
  Call Extruder 0.32322
  MoveL (T16130) to (118.06, 111.31, 17.5) mm, rotated rx 180 ry 0 rz -180 deg; joints [3.26, 68.93, -33.334, 5.588, -35.726, -4.542]
  Call Extruder 0.00328
  MoveL (T16131) to (117.97, 111.37, 17.5) mm, rotated rx 180 ry 0 rz -180 deg; joints [2.362, 71.224, -37.647, 4.266, -33.65, -3.553]
  Call Extruder 0.01316
  MoveL (T16132) to (117.54, 111.37, 17.5) mm, rotated rx 180 ry 0 rz -180 deg; joints [2.362, 71.224, -37.647, 4.266, -33.65, -3.553]
  Call Extruder 0.32579
  MoveL (T16133) to (110.01, 103.84, 17.5) mm, rotated rx 180 ry 0 rz -180 deg; joints [2.246, 71.21, -37.621, 4.055, -33.656, -3.377]
  Call Extruder 0.0177
  MoveL (T16134) to (109.44, 103.84, 17.5) mm, rotated rx 180 ry 0 rz -180 deg; joints [2.246, 71.21, -37.621, 4.055, -33.656, -3.377]
  Call Extruder 0.32579
  MoveL (T16135) to (116.96, 111.37, 17.5) mm, rotated rx 180 ry 0 rz -180 deg; joints [1.417, 68.731, -32.958, 2.423, -35.796, -1.966]
  Call Extruder 0.01118
  MoveL (T16136) to (116.6, 111.37, 17.5) mm, rotated rx 180 ry 0 rz -180 deg; joints [1.417, 68.731, -32.958, 2.423, -35.796, -1.966]
  Call Extruder 0.015
  MoveL (T16137) to (116.82, 111.81, 17.5) mm, rotated rx 180 ry 0 rz -180 deg; joints [1.417, 68.731, -32.958, 2.423, -35.796, -1.966]
  Call Extruder 0.34467
  MoveL (T16138) to (108.86, 103.84, 17.5) mm, rotated rx 180 ry 0 rz -180 deg; joints [1.417, 68.731, -32.958, 2.423, -35.796, -1.966]
  Call Extruder 0.0177
  MoveL (T16139) to (108.28, 103.84, 17.5) mm, rotated rx 180 ry 0 rz -180 deg; joints [1.42, 68.419, -32.373, 2.412, -36.07, -1.95]
  Call Extruder 0.39594
  MoveL (T16140) to (117.43, 112.99, 17.5) mm, rotated rx 180 ry 0 rz -180 deg; joints [2.319, 66.326, -28.439, 3.773, -37.947, -2.977]
  Call Extruder 0.04072
  MoveL (T16141) to (118.03, 114.18, 17.5) mm, rotated rx 180 ry 0 rz -180 deg; joints [2.319, 66.326, -28.439, 3.773, -37.947, -2.977]
  Call Extruder 0.4472
  MoveL (T16142) to (107.7, 103.84, 17.5) mm, rotated rx 180 ry 0 rz -180 deg; joints [2.319, 66.326, -28.439, 3.773, -37.947, -2.977]
  Call Extruder 0.0177
  MoveL (T16143) to (107.12, 103.84, 17.5) mm, rotated rx 180 ry 0 rz -180 deg; joints [1.941, 66.293, -28.377, 3.156, -37.958, -2.49]
  Call Extruder 0.49847
  MoveL (T16144) to (118.64, 115.36, 17.5) mm, rotated rx 180 ry 0 rz -180 deg; joints [1.941, 66.293, -28.377, 3.156, -37.958, -2.49]
  Call Extruder 0.04072
  MoveL (T16145) to (119.25, 116.55, 17.5) mm, rotated rx 180 ry 0 rz -180 deg; joints [3.239, 69.942, -35.237, 5.675, -34.837, -4.663]
  Call Extruder 0.54539
  MoveL (T16146) to (106.64, 103.94, 17.5) mm, rotated rx 180 ry 0 rz -180 deg; joints [3.239, 69.942, -35.237, 5.675, -34.837, -4.663]
  Call Extruder 0.01252
  MoveL (T16147) to (106.36, 104.23, 17.5) mm, rotated rx 180 ry 0 rz -180 deg; joints [3.239, 69.942, -35.237, 5.675, -34.837, -4.663]
  Call Extruder 0.57634
  MoveL (T16148) to (119.67, 117.55, 17.5) mm, rotated rx 180 ry 0 rz -180 deg; joints [3.232, 70.274, -35.86, 5.706, -34.547, -4.704]
  Call Extruder 0.01389
  MoveL (T16149) to (119.78, 117.99, 17.5) mm, rotated rx 180 ry 0 rz -180 deg; joints [3.232, 70.274, -35.86, 5.706, -34.547, -4.704]
  Call Extruder 0.00751
  MoveL (T16150) to (119.78, 118.24, 17.5) mm, rotated rx 180 ry 0 rz -180 deg; joints [3.232, 70.274, -35.86, 5.706, -34.547, -4.704]
  Call Extruder 0.59354
  MoveL (T16151) to (106.07, 104.52, 17.5) mm, rotated rx 180 ry 0 rz -180 deg; joints [2.845, 71.29, -37.771, 5.143, -33.626, -4.286]
  Call Extruder 0.01252
  MoveL (T16152) to (105.78, 104.81, 17.5) mm, rotated rx 180 ry 0 rz -180 deg; joints [2.845, 71.29, -37.771, 5.143, -33.626, -4.286]
  Call Extruder 0.60606
  MoveL (T16153) to (119.78, 118.81, 17.5) mm, rotated rx 180 ry 0 rz -180 deg; joints [2.729, 71.273, -37.739, 4.931, -33.632, -4.109]
  Call Extruder 0.0177
  MoveL (T16154) to (119.78, 119.39, 17.5) mm, rotated rx 180 ry 0 rz -180 deg; joints [2.729, 71.273, -37.739, 4.931, -33.632, -4.109]
  Call Extruder 0.6185
  MoveL (T16155) to (105.49, 105.1, 17.5) mm, rotated rx 180 ry 0 rz -180 deg; joints [2.729, 71.273, -37.739, 4.931, -33.632, -4.109]
  Call Extruder 0.0015
  MoveL (T16156) to (105.47, 105.15, 17.5) mm, rotated rx 180 ry 0 rz -180 deg; joints [1.429, 67.465, -30.58, 2.38, -36.909, -1.904]
  Call Extruder 0.01574
  MoveL (T16157) to (105.47, 105.66, 17.5) mm, rotated rx 180 ry 0 rz -180 deg; joints [1.429, 67.465, -30.58, 2.38, -36.909, -1.904]
  Call Extruder 0.61932
  MoveL (T16158) to (119.78, 119.97, 17.5) mm, rotated rx 180 ry 0 rz -180 deg; joints [1.432, 67.169, -30.023, 2.371, -37.169, -1.89]
  Call Extruder 0.00627
  MoveL (T16159) to (119.78, 120.18, 17.5) mm, rotated rx 180 ry 0 rz -180 deg; joints [1.432, 67.169, -30.023, 2.371, -37.169, -1.89]
  Call Extruder 0.00169
  MoveL (T16160) to (119.76, 120.23, 17.5) mm, rotated rx 180 ry 0 rz -180 deg; joints [1.432, 67.169, -30.023, 2.371, -37.169, -1.89]
  Call Extruder 0.00653
  MoveL (T16161) to (119.61, 120.38, 17.5) mm, rotated rx 180 ry 0 rz -180 deg; joints [1.821, 66.283, -28.359, 2.96, -37.961, -2.335]
  Call Extruder 0.61188
  MoveL (T16162) to (105.47, 106.24, 17.5) mm, rotated rx 180 ry 0 rz -180 deg; joints [1.821, 66.283, -28.359, 2.96, -37.961, -2.335]
  Call Extruder 0.0177
  MoveL (T16163) to (105.47, 106.82, 17.5) mm, rotated rx 180 ry 0 rz -180 deg; joints [1.442, 66.258, -28.311, 2.344, -37.97, -1.848]
  Call Extruder 0.59936
  MoveL (T16164) to (119.32, 120.67, 17.5) mm, rotated rx 180 ry 0 rz -180 deg; joints [1.442, 66.258, -28.311, 2.344, -37.97, -1.848]
  Call Extruder 0.01252
  MoveL (T16165) to (119.03, 120.96, 17.5) mm, rotated rx 180 ry 0 rz -180 deg; joints [3.211, 71.348, -37.88, 5.809, -33.604, -4.843]
  Call Extruder 0.58584
  MoveL (T16166) to (105.49, 107.42, 17.5) mm, rotated rx 180 ry 0 rz -180 deg; joints [3.211, 71.348, -37.88, 5.809, -33.604, -4.843]
  Call Extruder 0.02102
  MoveL (T16167) to (105.65, 108.09, 17.5) mm, rotated rx 180 ry 0 rz -180 deg; joints [3.211, 71.348, -37.88, 5.809, -33.604, -4.843]
  Call Extruder 0.0048
  MoveL (T16168) to (105.72, 108.23, 17.5) mm, rotated rx 180 ry 0 rz -180 deg; joints [3.226, 70.592, -36.458, 5.735, -34.268, -4.745]
  Call Extruder 0.55945
  MoveL (T16169) to (118.65, 121.16, 17.5) mm, rotated rx 180 ry 0 rz -180 deg; joints [3.226, 70.592, -36.458, 5.735, -34.268, -4.745]
  Call Extruder 0.0177
  MoveL (T16170) to (118.07, 121.16, 17.5) mm, rotated rx 180 ry 0 rz -180 deg; joints [3.226, 70.592, -36.458, 5.735, -34.268, -4.745]
  Call Extruder 0.50836
  MoveL (T16171) to (106.33, 109.41, 17.5) mm, rotated rx 180 ry 0 rz -180 deg; joints [3.226, 70.592, -36.458, 5.735, -34.268, -4.745]
  Call Extruder 0.04056
  MoveL (T16172) to (106.93, 110.59, 17.5) mm, rotated rx 180 ry 0 rz -180 deg; joints [3.226, 70.592, -36.458, 5.735, -34.268, -4.745]
  Call Extruder 0.45726
  MoveL (T16173) to (117.49, 121.16, 17.5) mm, rotated rx 180 ry 0 rz -180 deg; joints [3.226, 70.592, -36.458, 5.735, -34.268, -4.745]
  Call Extruder 0.0177
  MoveL (T16174) to (116.92, 121.16, 17.5) mm, rotated rx 180 ry 0 rz -180 deg; joints [3.226, 70.592, -36.458, 5.735, -34.268, -4.745]
  Call Extruder 0.40616
  MoveL (T16175) to (107.53, 111.77, 17.5) mm, rotated rx 180 ry 0 rz -180 deg; joints [3.226, 70.592, -36.458, 5.735, -34.268, -4.745]
  Call Extruder 0.04056
  MoveL (T16176) to (108.13, 112.95, 17.5) mm, rotated rx 180 ry 0 rz -180 deg; joints [3.226, 70.592, -36.458, 5.735, -34.268, -4.745]
  Call Extruder 0.35507
  MoveL (T16177) to (116.34, 121.16, 17.5) mm, rotated rx 180 ry 0 rz -180 deg; joints [3.226, 70.592, -36.458, 5.735, -34.268, -4.745]
  Call Extruder 0.0177
  MoveL (T16178) to (115.76, 121.16, 17.5) mm, rotated rx 180 ry 0 rz -180 deg; joints [3.226, 70.592, -36.458, 5.735, -34.268, -4.745]
  Call Extruder 0.31171
  MoveL (T16179) to (108.56, 113.95, 17.5) mm, rotated rx 180 ry 0 rz -180 deg; joints [3.219, 70.919, -37.073, 5.767, -33.981, -4.787]
  Call Extruder 0.0177
  MoveL (T16180) to (107.98, 113.95, 17.5) mm, rotated rx 180 ry 0 rz -180 deg; joints [3.219, 70.919, -37.073, 5.767, -33.981, -4.787]
  Call Extruder 0.31171
  MoveL (T16181) to (115.18, 121.16, 17.5) mm, rotated rx 180 ry 0 rz -180 deg; joints [3.219, 70.919, -37.073, 5.767, -33.981, -4.787]
  Call Extruder 0.0177
  MoveL (T16182) to (114.6, 121.16, 17.5) mm, rotated rx 180 ry 0 rz -180 deg; joints [3.219, 70.919, -37.073, 5.767, -33.981, -4.787]
  Call Extruder 0.30914
  MoveL (T16183) to (107.46, 114.01, 17.5) mm, rotated rx 180 ry 0 rz -180 deg; joints [3.219, 70.919, -37.073, 5.767, -33.981, -4.787]
  Call Extruder 0.01252
  MoveL (T16184) to (107.17, 114.3, 17.5) mm, rotated rx 180 ry 0 rz -180 deg; joints [3.219, 70.919, -37.073, 5.767, -33.981, -4.787]
  Call Extruder 0.29663
  MoveL (T16185) to (114.02, 121.16, 17.5) mm, rotated rx 180 ry 0 rz -180 deg; joints [3.219, 70.919, -37.073, 5.767, -33.981, -4.787]
  Call Extruder 0.0177
  MoveL (T16186) to (113.44, 121.16, 17.5) mm, rotated rx 180 ry 0 rz -180 deg; joints [1.407, 66.146, -28.509, 2.304, -37.66, -1.824]
  Call Extruder 0.28411
  MoveL (T16187) to (106.88, 114.59, 17.5) mm, rotated rx 180 ry 0 rz -180 deg; joints [1.407, 66.359, -28.543, 2.294, -37.839, -1.812]
  Call Extruder 0.01252
  MoveL (T16188) to (106.59, 114.88, 17.5) mm, rotated rx 180 ry 0 rz -180 deg; joints [1.407, 66.359, -28.543, 2.294, -37.839, -1.812]
  Call Extruder 0.2716
  MoveL (T16189) to (112.87, 121.16, 17.5) mm, rotated rx 180 ry 0 rz -180 deg; joints [1.407, 66.359, -28.543, 2.294, -37.839, -1.812]
  Call Extruder 0.0177
  MoveL (T16190) to (112.29, 121.16, 17.5) mm, rotated rx 180 ry 0 rz -180 deg; joints [1.407, 66.359, -28.543, 2.294, -37.839, -1.812]
  Call Extruder 0.25908
  MoveL (T16191) to (106.3, 115.17, 17.5) mm, rotated rx 180 ry 0 rz -180 deg; joints [1.407, 66.359, -28.543, 2.294, -37.839, -1.812]
  Call Extruder 0.01252
  MoveL (T16192) to (106.01, 115.46, 17.5) mm, rotated rx 180 ry 0 rz -180 deg; joints [1.407, 66.359, -28.543, 2.294, -37.839, -1.812]
  Call Extruder 0.24657
  MoveL (T16193) to (111.71, 121.16, 17.5) mm, rotated rx 180 ry 0 rz -180 deg; joints [1.407, 66.359, -28.543, 2.294, -37.839, -1.812]
  Call Extruder 0.0177
  MoveL (T16194) to (111.13, 121.16, 17.5) mm, rotated rx 180 ry 0 rz -180 deg; joints [1.407, 66.359, -28.543, 2.294, -37.839, -1.812]
  Call Extruder 0.23405
  MoveL (T16195) to (105.72, 115.75, 17.5) mm, rotated rx 180 ry 0 rz -180 deg; joints [1.407, 66.359, -28.543, 2.294, -37.839, -1.812]
  Call Extruder 0.00641
  MoveL (T16196) to (105.58, 115.9, 17.5) mm, rotated rx 180 ry 0 rz -180 deg; joints [1.407, 66.359, -28.543, 2.294, -37.839, -1.812]
  Call Extruder 0.00169
  MoveL (T16197) to (105.55, 115.95, 17.5) mm, rotated rx 180 ry 0 rz -180 deg; joints [1.407, 66.359, -28.543, 2.294, -37.839, -1.812]
  Call Extruder 0.00643
  MoveL (T16198) to (105.55, 116.16, 17.5) mm, rotated rx 180 ry 0 rz -180 deg; joints [1.363, 71.199, -37.64, 2.465, -33.584, -2.054]
  Call Extruder 0.21634
  MoveL (T16199) to (110.55, 121.16, 17.5) mm, rotated rx 180 ry 0 rz -180 deg; joints [1.363, 71.199, -37.64, 2.465, -33.584, -2.054]
  Call Extruder 0.0177
  MoveL (T16200) to (109.97, 121.16, 17.5) mm, rotated rx 180 ry 0 rz -180 deg; joints [3.241, 71.426, -38.067, 5.88, -33.499, -4.909]
  Call Extruder 0.19131
  MoveL (T16201) to (105.55, 116.73, 17.5) mm, rotated rx 180 ry 0 rz -180 deg; joints [3.241, 71.426, -38.067, 5.88, -33.499, -4.909]
  Call Extruder 0.0177
  MoveL (T16202) to (105.55, 117.31, 17.5) mm, rotated rx 180 ry 0 rz -180 deg; joints [3.351, 66.345, -28.516, 5.454, -37.955, -4.305]
  Call Extruder 0.16628
  MoveL (T16203) to (109.4, 121.16, 17.5) mm, rotated rx 180 ry 0 rz -180 deg; joints [1.409, 66.154, -28.157, 2.289, -38.019, -1.803]
  Call Extruder 0.0177
  MoveL (T16204) to (108.82, 121.16, 17.5) mm, rotated rx 180 ry 0 rz -180 deg; joints [1.409, 66.154, -28.157, 2.289, -38.019, -1.803]
  Call Extruder 0.14125
  MoveL (T16205) to (105.55, 117.89, 17.5) mm, rotated rx 180 ry 0 rz -180 deg; joints [1.407, 66.344, -28.514, 2.294, -37.853, -1.812]
  Call Extruder 0.0177
  MoveL (T16206) to (105.55, 118.47, 17.5) mm, rotated rx 180 ry 0 rz -180 deg; joints [1.365, 66.15, -28.149, 2.217, -38.022, -1.747]
  Call Extruder 0.11622
  MoveL (T16207) to (108.24, 121.16, 17.5) mm, rotated rx 180 ry 0 rz -180 deg; joints [1.365, 66.15, -28.149, 2.217, -38.022, -1.747]
  Call Extruder 0.0177
  MoveL (T16208) to (107.66, 121.16, 17.5) mm, rotated rx 180 ry 0 rz -180 deg; joints [1.365, 66.15, -28.149, 2.217, -38.022, -1.747]
  Call Extruder 0.09119
  MoveL (T16209) to (105.55, 119.05, 17.5) mm, rotated rx 180 ry 0 rz -180 deg; joints [1.365, 66.15, -28.149, 2.217, -38.022, -1.747]
  Call Extruder 0.0177
  MoveL (T16210) to (105.55, 119.63, 17.5) mm, rotated rx 180 ry 0 rz -180 deg; joints [1.365, 66.15, -28.149, 2.217, -38.022, -1.747]
  Call Extruder 0.06616
  MoveL (T16211) to (107.08, 121.16, 17.5) mm, rotated rx 180 ry 0 rz -180 deg; joints [1.319, 71.324, -37.875, 2.393, -33.473, -1.996]
  Call Extruder 0.0177
  MoveL (T16212) to (106.5, 121.16, 17.5) mm, rotated rx 180 ry 0 rz -180 deg; joints [1.319, 71.324, -37.875, 2.393, -33.473, -1.996]
  Call Extruder 0.04905
  MoveL (T16213) to (105.37, 120.02, 17.5) mm, rotated rx 180 ry 0 rz -180 deg; joints [1.319, 71.324, -37.875, 2.393, -33.473, -1.996]
  Set speed (45.0 mm/s)
  Call Extruder -1.6
  MoveL (T16214) to (105.37, 120.02, 17.5) mm, rotated rx 180 ry 0 rz -180 deg; joints [3.282, 71.563, -38.324, 5.971, -33.383, -4.992]
  Set speed (120.0 mm/s)
  MoveL (T16215) to (105.37, 120.02, 17.5) mm, rotated rx 180 ry 0 rz -180 deg; joints [3.282, 71.563, -38.324, 5.971, -33.383, -4.992]
  Call Extruder -0.38
  MoveL (T16216) to (106.12, 120.78, 17.5) mm, rotated rx 180 ry 0 rz -180 deg; joints [3.398, 66.247, -28.331, 5.519, -38.045, -4.351]
  Set speed (45.0 mm/s)
  Call Extruder -0.02
  MoveL (T16217) to (106.12, 120.78, 17.5) mm, rotated rx 180 ry 0 rz -180 deg; joints [3.398, 66.247, -28.331, 5.519, -38.045, -4.351]
  Set speed (150.0 mm/s)
  MoveL (T16218) to (106.12, 120.78, 19.5) mm, rotated rx 180 ry 0 rz -180 deg; joints [3.398, 66.247, -28.331, 5.519, -38.045, -4.351]
  MoveL (T16219) to (120.05, 117.4, 19.5) mm, rotated rx 180 ry 0 rz -180 deg; joints [1.366, 66.048, -27.957, 2.214, -38.111, -1.742]
  MoveL (T16220) to (120.05, 117.4, 17.5) mm, rotated rx 180 ry 0 rz -180 deg; joints [1.366, 66.048, -27.957, 2.214, -38.111, -1.742]
  Set speed (40.0 mm/s)
  Call Extruder 2.0
  MoveL (T16221) to (120.05, 117.4, 17.5) mm, rotated rx 180 ry 0 rz -180 deg; joints [1.365, 66.134, -28.12, 2.216, -38.035, -1.746]
  Set speed (50.0 mm/s)
  MoveL (T16222) to (120.05, 117.4, 17.5) mm, rotated rx 180 ry 0 rz -180 deg; joints [1.365, 66.134, -28.12, 2.216, -38.035, -1.746]
  Call Extruder 0.01089
  MoveL (T16223) to (119.96, 117.05, 17.5) mm, rotated rx 180 ry 0 rz -180 deg; joints [1.365, 66.134, -28.12, 2.216, -38.035, -1.746]
  Call Extruder 0.0635
  MoveL (T16224) to (119.01, 115.2, 17.5) mm, rotated rx 180 ry 0 rz -180 deg; joints [1.365, 66.134, -28.12, 2.216, -38.035, -1.746]
  Call Extruder 0.09231
  MoveL (T16225) to (121.16, 113.06, 17.5) mm, rotated rx 180 ry 0 rz -180 deg; joints [1.332, 65.942, -27.759, 2.155, -38.203, -1.694]
  Call Extruder 0.03385
  MoveL (T16226) to (121.16, 111.94, 17.5) mm, rotated rx 180 ry 0 rz -180 deg; joints [1.332, 65.942, -27.759, 2.155, -38.203, -1.694]
  Call Extruder 0.06789
  MoveL (T16227) to (119.58, 110.37, 17.5) mm, rotated rx 180 ry 0 rz -180 deg; joints [1.332, 65.942, -27.759, 2.155, -38.203, -1.694]
  Call Extruder 0.03053
  MoveL (T16228) to (120.29, 109.66, 17.5) mm, rotated rx 180 ry 0 rz -180 deg; joints [1.332, 65.942, -27.759, 2.155, -38.203, -1.694]
  Call Extruder 0.00661
  MoveL (T16229) to (120.37, 109.46, 17.5) mm, rotated rx 180 ry 0 rz -180 deg; joints [1.332, 65.942, -27.759, 2.155, -38.203, -1.694]
  Call Extruder 0.00686
  MoveL (T16230) to (120.37, 109.23, 17.5) mm, rotated rx 180 ry 0 rz -180 deg; joints [1.332, 65.942, -27.759, 2.155, -38.203, -1.694]
  Call Extruder 0.03378
  MoveL (T16231) to (121.16, 108.45, 17.5) mm, rotated rx 180 ry 0 rz -180 deg; joints [1.332, 65.942, -27.759, 2.155, -38.203, -1.694]
  Call Extruder 0.03385
  MoveL (T16232) to (121.16, 107.34, 17.5) mm, rotated rx 180 ry 0 rz -180 deg; joints [1.332, 65.942, -27.759, 2.155, -38.203, -1.694]
  Call Extruder 0.03378
  MoveL (T16233) to (120.37, 106.56, 17.5) mm, rotated rx 180 ry 0 rz -180 deg; joints [1.323, 65.942, -27.758, 2.14, -38.203, -1.682]
  Call Extruder 0.04531
  MoveL (T16234) to (120.37, 105.07, 17.5) mm, rotated rx 180 ry 0 rz -180 deg; joints [1.323, 65.942, -27.758, 2.14, -38.203, -1.682]
  Call Extruder 0.00661
  MoveL (T16235) to (120.29, 104.87, 17.5) mm, rotated rx 180 ry 0 rz -180 deg; joints [1.323, 65.942, -27.758, 2.14, -38.203, -1.682]
  Call Extruder 0.00334
  MoveL (T16236) to (120.21, 104.79, 17.5) mm, rotated rx 180 ry 0 rz -180 deg; joints [1.276, 71.45, -38.111, 2.321, -33.36, -1.939]
  Call Extruder 0.04071
  MoveL (T16237) to (121.16, 103.84, 17.5) mm, rotated rx 180 ry 0 rz -180 deg; joints [1.276, 71.45, -38.111, 2.321, -33.36, -1.939]
  Call Extruder 0.07441
  MoveL (T16238) to (121.16, 106.29, 17.5) mm, rotated rx 180 ry 0 rz -180 deg; joints [3.322, 71.701, -38.582, 6.063, -33.266, -5.076]
  Set speed (45.0 mm/s)
  Call Extruder -1.6
  MoveL (T16239) to (121.16, 106.29, 17.5) mm, rotated rx 180 ry 0 rz -180 deg; joints [3.322, 71.701, -38.582, 6.063, -33.266, -5.076]
  Set speed (120.0 mm/s)
  MoveL (T16240) to (121.16, 106.29, 17.5) mm, rotated rx 180 ry 0 rz -180 deg; joints [3.445, 66.149, -28.147, 5.584, -38.134, -4.397]
  Call Extruder -0.38
  MoveL (T16241) to (121.16, 105.22, 17.5) mm, rotated rx 180 ry 0 rz -180 deg; joints [3.445, 66.149, -28.147, 5.584, -38.134, -4.397]
  Set speed (45.0 mm/s)
  Call Extruder -0.02
  MoveL (T16242) to (121.16, 105.22, 17.5) mm, rotated rx 180 ry 0 rz -180 deg; joints [1.339, 65.943, -27.76, 2.165, -38.203, -1.702]
  Set speed (150.0 mm/s)
  MoveL (T16243) to (121.16, 105.22, 19.5) mm, rotated rx 180 ry 0 rz -180 deg; joints [1.339, 65.943, -27.76, 2.165, -38.203, -1.702]
  MoveL (T16244) to (119.44, 110.51, 19.5) mm, rotated rx 180 ry 0 rz -180 deg; joints [1.326, 65.957, -27.787, 2.145, -38.19, -1.686]
  MoveL (T16245) to (119.44, 110.51, 17.5) mm, rotated rx 180 ry 0 rz -180 deg; joints [1.326, 65.957, -27.787, 2.145, -38.19, -1.686]
  Set speed (40.0 mm/s)
  Call Extruder 2.0
  MoveL (T16246) to (119.44, 110.51, 17.5) mm, rotated rx 180 ry 0 rz -180 deg; joints [1.326, 65.957, -27.787, 2.145, -38.19, -1.686]
  Set speed (50.0 mm/s)
  MoveL (T16247) to (119.44, 110.51, 17.5) mm, rotated rx 180 ry 0 rz -180 deg; joints [1.326, 65.957, -27.787, 2.145, -38.19, -1.686]
  Call Extruder 0.05098
  MoveL (T16248) to (118.25, 111.7, 17.5) mm, rotated rx 180 ry 0 rz -180 deg; joints [1.326, 65.957, -27.787, 2.145, -38.19, -1.686]
  Call Extruder 0.00661
  MoveL (T16249) to (118.05, 111.78, 17.5) mm, rotated rx 180 ry 0 rz -180 deg; joints [1.326, 65.957, -27.787, 2.145, -38.19, -1.686]
  Call Extruder 0.00686
  MoveL (T16250) to (117.83, 111.78, 17.5) mm, rotated rx 180 ry 0 rz -180 deg; joints [1.326, 65.957, -27.787, 2.145, -38.19, -1.686]
  Call Extruder 0.01607
  MoveL (T16251) to (117.45, 112.15, 17.5) mm, rotated rx 180 ry 0 rz -180 deg; joints [1.326, 65.957, -27.787, 2.145, -38.19, -1.686]
  Call Extruder 0.04881
  MoveL (T16252) to (118.18, 113.58, 17.5) mm, rotated rx 180 ry 0 rz -180 deg; joints [1.326, 65.957, -27.787, 2.145, -38.19, -1.686]
  Call Extruder 0.12804
  MoveL (T16253) to (121.16, 116.55, 17.5) mm, rotated rx 180 ry 0 rz -180 deg; joints [1.326, 65.957, -27.787, 2.145, -38.19, -1.686]
  Call Extruder 0.03385
  MoveL (T16254) to (121.16, 117.66, 17.5) mm, rotated rx 180 ry 0 rz -180 deg; joints [1.326, 65.957, -27.787, 2.145, -38.19, -1.686]
  Call Extruder 0.04175
  MoveL (T16255) to (120.19, 118.63, 17.5) mm, rotated rx 180 ry 0 rz -180 deg; joints [1.323, 65.942, -27.758, 2.14, -38.203, -1.682]
  Call Extruder 0.04741
  MoveL (T16256) to (120.19, 120.19, 17.5) mm, rotated rx 180 ry 0 rz -180 deg; joints [1.323, 65.942, -27.758, 2.14, -38.203, -1.682]
  Call Extruder 0.04175
  MoveL (T16257) to (121.16, 121.16, 17.5) mm, rotated rx 180 ry 0 rz -180 deg; joints [1.323, 65.942, -27.758, 2.14, -38.203, -1.682]
  Call Extruder 0.07441
  MoveL (T16258) to (121.16, 118.71, 17.5) mm, rotated rx 180 ry 0 rz -180 deg; joints [1.321, 66.177, -28.2, 2.146, -37.997, -1.691]
  Set speed (45.0 mm/s)
  Call Extruder -1.6
  MoveL (T16259) to (121.16, 118.71, 17.5) mm, rotated rx 180 ry 0 rz -180 deg; joints [1.321, 66.177, -28.2, 2.146, -37.997, -1.691]
  Set speed (120.0 mm/s)
  MoveL (T16260) to (121.16, 118.71, 17.5) mm, rotated rx 180 ry 0 rz -180 deg; joints [1.321, 66.177, -28.2, 2.146, -37.997, -1.691]
  Call Extruder -0.38
  MoveL (T16261) to (121.16, 119.78, 17.5) mm, rotated rx 180 ry 0 rz -180 deg; joints [1.321, 66.177, -28.2, 2.146, -37.997, -1.691]
  Set speed (45.0 mm/s)
  Call Extruder -0.02
  MoveL (T16262) to (121.16, 119.78, 17.5) mm, rotated rx 180 ry 0 rz -180 deg; joints [1.321, 66.177, -28.2, 2.146, -37.997, -1.691]
  Set speed (150.0 mm/s)
  MoveL (T16263) to (121.16, 119.78, 19.5) mm, rotated rx 180 ry 0 rz -180 deg; joints [1.321, 66.177, -28.2, 2.146, -37.997, -1.691]
  MoveL (T16264) to (104.34, 103.54, 19.5) mm, rotated rx 180 ry 0 rz -180 deg; joints [1.321, 66.177, -28.2, 2.146, -37.997, -1.691]
  MoveL (T16265) to (104.34, 103.54, 17.7) mm, rotated rx 180 ry 0 rz -180 deg; joints [1.321, 66.177, -28.2, 2.146, -37.997, -1.691]
  Set speed (40.0 mm/s)
  Call Extruder 2.0
  MoveL (T16266) to (104.34, 103.54, 17.7) mm, rotated rx 180 ry 0 rz -180 deg; joints [1.321, 66.177, -28.2, 2.146, -37.997, -1.691]
  Call Extruder 0.52159
  MoveL (T16267) to (121.46, 103.54, 17.7) mm, rotated rx 180 ry 0 rz -180 deg; joints [1.402, 70.356, -36.054, 2.487, -34.327, -2.054]
  Call Extruder 0.54596
  MoveL (T16268) to (121.46, 121.46, 17.7) mm, rotated rx 180 ry 0 rz -180 deg; joints [1.402, 70.356, -36.054, 2.487, -34.327, -2.054]
  Call Extruder 0.54596
  MoveL (T16269) to (103.54, 121.46, 17.7) mm, rotated rx 180 ry 0 rz -180 deg; joints [1.402, 70.356, -36.054, 2.487, -34.327, -2.054]
  Call Extruder 0.54596
  MoveL (T16270) to (103.54, 103.54, 17.7) mm, rotated rx 180 ry 0 rz -180 deg; joints [1.402, 70.356, -36.054, 2.487, -34.327, -2.054]
  Call Extruder 0.02254
  MoveL (T16271) to (104.28, 103.54, 17.7) mm, rotated rx 180 ry 0 rz -180 deg; joints [1.402, 70.356, -36.054, 2.487, -34.327, -2.054]
  Set speed (150.0 mm/s)
  MoveL (T16272) to (103.53, 103.13, 17.7) mm, rotated rx 180 ry 0 rz -180 deg; joints [1.402, 70.356, -36.054, 2.487, -34.327, -2.054]
  Set speed (40.0 mm/s)
  MoveL (T16273) to (103.53, 103.13, 17.7) mm, rotated rx 180 ry 0 rz -180 deg; joints [1.402, 70.356, -36.054, 2.487, -34.327, -2.054]
  Call Extruder 0.55858
  MoveL (T16274) to (121.87, 103.13, 17.7) mm, rotated rx 180 ry 0 rz -180 deg; joints [1.402, 70.356, -36.054, 2.487, -34.327, -2.054]
  Call Extruder 0.57077
  MoveL (T16275) to (121.87, 121.87, 17.7) mm, rotated rx 180 ry 0 rz -180 deg; joints [1.402, 70.356, -36.054, 2.487, -34.327, -2.054]
  Call Extruder 0.57077
  MoveL (T16276) to (103.13, 121.87, 17.7) mm, rotated rx 180 ry 0 rz -180 deg; joints [1.402, 70.356, -36.054, 2.487, -34.327, -2.054]
  Call Extruder 0.57077
  MoveL (T16277) to (103.13, 103.13, 17.7) mm, rotated rx 180 ry 0 rz -180 deg; joints [1.396, 71.106, -37.465, 2.519, -33.667, -2.097]
  Call Extruder 0.01036
  MoveL (T16278) to (103.47, 103.13, 17.7) mm, rotated rx 180 ry 0 rz -180 deg; joints [1.396, 71.106, -37.465, 2.519, -33.667, -2.097]
  Set speed (150.0 mm/s)
  MoveL (T16279) to (102.72, 102.81, 17.7) mm, rotated rx 180 ry 0 rz -180 deg; joints [1.396, 71.106, -37.465, 2.519, -33.667, -2.097]
  Set speed (25.0 mm/s)
  MoveL (T16280) to (102.72, 102.81, 17.7) mm, rotated rx 180 ry 0 rz -180 deg; joints [3.316, 66.419, -28.655, 5.405, -37.888, -4.27]
  Call Extruder 0.00259
  MoveL (T16281) to (102.72, 102.72, 17.7) mm, rotated rx 180 ry 0 rz -180 deg; joints [3.316, 66.419, -28.655, 5.405, -37.888, -4.27]
  Call Extruder 0.59557
  MoveL (T16282) to (122.28, 102.72, 17.7) mm, rotated rx 180 ry 0 rz -180 deg; joints [3.316, 66.419, -28.655, 5.405, -37.888, -4.27]
  Call Extruder 0.59557
  MoveL (T16283) to (122.28, 122.28, 17.7) mm, rotated rx 180 ry 0 rz -180 deg; joints [2.938, 66.37, -28.562, 4.786, -37.905, -3.78]
  Call Extruder 0.59557
  MoveL (T16284) to (102.72, 122.28, 17.7) mm, rotated rx 180 ry 0 rz -180 deg; joints [2.938, 66.37, -28.562, 4.786, -37.905, -3.78]
  Call Extruder 0.59115
  MoveL (T16285) to (102.72, 102.87, 17.7) mm, rotated rx 180 ry 0 rz -180 deg; joints [2.938, 66.37, -28.562, 4.786, -37.905, -3.78]
  Set speed (150.0 mm/s)
  MoveL (T16286) to (102.78, 102.75, 17.7) mm, rotated rx 180 ry 0 rz -180 deg; joints [2.938, 66.37, -28.562, 4.786, -37.905, -3.78]
  Set speed (45.0 mm/s)
  Call Extruder -1.6
  MoveL (T16287) to (102.78, 102.75, 17.7) mm, rotated rx 180 ry 0 rz -180 deg; joints [3.295, 67.335, -30.376, 5.469, -37.085, -4.368]
  Set speed (120.0 mm/s)
  MoveL (T16288) to (102.78, 102.75, 17.7) mm, rotated rx 180 ry 0 rz -180 deg; joints [3.295, 67.335, -30.376, 5.469, -37.085, -4.368]
  Call Extruder -0.05166
  MoveL (T16289) to (102.72, 102.72, 17.7) mm, rotated rx 180 ry 0 rz -180 deg; joints [3.288, 67.633, -30.936, 5.491, -36.823, -4.4]
  Call Extruder -0.32834
  MoveL (T16290) to (103.65, 102.72, 17.7) mm, rotated rx 180 ry 0 rz -180 deg; joints [3.288, 67.633, -30.936, 5.491, -36.823, -4.4]
  Set speed (45.0 mm/s)
  Call Extruder -0.02
  MoveL (T16291) to (103.65, 102.72, 17.7) mm, rotated rx 180 ry 0 rz -180 deg; joints [3.288, 67.633, -30.936, 5.491, -36.823, -4.4]
  Set speed (150.0 mm/s)
  MoveL (T16292) to (103.65, 102.72, 19.7) mm, rotated rx 180 ry 0 rz -180 deg; joints [1.879, 71.147, -37.542, 3.393, -33.652, -2.825]
  MoveL (T16293) to (106.08, 103.93, 19.7) mm, rotated rx 180 ry 0 rz -180 deg; joints [1.879, 71.147, -37.542, 3.393, -33.652, -2.825]
  MoveL (T16294) to (106.08, 103.93, 17.7) mm, rotated rx 180 ry 0 rz -180 deg; joints [1.763, 71.136, -37.521, 3.182, -33.656, -2.649]
  Set speed (40.0 mm/s)
  Call Extruder 2.0
  MoveL (T16295) to (106.08, 103.93, 17.7) mm, rotated rx 180 ry 0 rz -180 deg; joints [1.763, 71.136, -37.521, 3.182, -33.656, -2.649]
  Set speed (50.0 mm/s)
  MoveL (T16296) to (106.08, 103.93, 17.7) mm, rotated rx 180 ry 0 rz -180 deg; joints [1.763, 71.136, -37.521, 3.182, -33.656, -2.649]
  Call Extruder 0.00361
  MoveL (T16297) to (106.17, 103.84, 17.7) mm, rotated rx 180 ry 0 rz -180 deg; joints [1.763, 71.136, -37.521, 3.182, -33.656, -2.649]
  Call Extruder 0.0708
  MoveL (T16298) to (103.84, 103.84, 17.7) mm, rotated rx 180 ry 0 rz -180 deg; joints [1.405, 70.04, -35.461, 2.474, -34.605, -2.037]
  Call Extruder 0.05255
  MoveL (T16299) to (105.06, 105.06, 17.7) mm, rotated rx 180 ry 0 rz -180 deg; joints [1.405, 70.04, -35.461, 2.474, -34.605, -2.037]
  Call Extruder 0.03217
  MoveL (T16300) to (105.06, 106.12, 17.7) mm, rotated rx 180 ry 0 rz -180 deg; joints [1.405, 70.04, -35.461, 2.474, -34.605, -2.037]
  Call Extruder 0.0525
  MoveL (T16301) to (103.84, 107.34, 17.7) mm, rotated rx 180 ry 0 rz -180 deg; joints [1.405, 70.04, -35.461, 2.474, -34.605, -2.037]
  Call Extruder 0.03385
  MoveL (T16302) to (103.84, 108.45, 17.7) mm, rotated rx 180 ry 0 rz -180 deg; joints [1.405, 70.04, -35.461, 2.474, -34.605, -2.037]
  Call Extruder 0.13495
  MoveL (T16303) to (106.98, 111.58, 17.7) mm, rotated rx 180 ry 0 rz -180 deg; joints [1.408, 69.712, -34.843, 2.462, -34.894, -2.019]
  Call Extruder 0.04156
  MoveL (T16304) to (107.6, 112.8, 17.7) mm, rotated rx 180 ry 0 rz -180 deg; joints [1.408, 69.712, -34.843, 2.462, -34.894, -2.019]
  Call Extruder 0.16166
  MoveL (T16305) to (103.84, 116.55, 17.7) mm, rotated rx 180 ry 0 rz -180 deg; joints [1.408, 69.712, -34.843, 2.462, -34.894, -2.019]
  Call Extruder 0.03385
  MoveL (T16306) to (103.84, 117.66, 17.7) mm, rotated rx 180 ry 0 rz -180 deg; joints [1.408, 69.712, -34.843, 2.462, -34.894, -2.019]
  Call Extruder 0.05612
  MoveL (T16307) to (105.15, 118.96, 17.7) mm, rotated rx 180 ry 0 rz -180 deg; joints [2.818, 66.356, -28.535, 4.59, -37.909, -3.624]
  Call Extruder 0.02709
  MoveL (T16308) to (105.15, 119.85, 17.7) mm, rotated rx 180 ry 0 rz -180 deg; joints [2.818, 66.356, -28.535, 4.59, -37.909, -3.624]
  Call Extruder 0.05612
  MoveL (T16309) to (103.84, 121.16, 17.7) mm, rotated rx 180 ry 0 rz -180 deg; joints [2.818, 66.356, -28.535, 4.59, -37.909, -3.624]
  Call Extruder 0.06345
  MoveL (T16310) to (105.93, 121.16, 17.7) mm, rotated rx 180 ry 0 rz -180 deg; joints [2.818, 66.356, -28.535, 4.59, -37.909, -3.624]
  Call Extruder 0.01096
  MoveL (T16311) to (105.67, 120.9, 17.7) mm, rotated rx 180 ry 0 rz -180 deg; joints [2.44, 66.314, -28.458, 3.972, -37.923, -3.135]
  Set speed (45.0 mm/s)
  Call Extruder -1.6
  MoveL (T16312) to (105.67, 120.9, 17.7) mm, rotated rx 180 ry 0 rz -180 deg; joints [2.44, 66.314, -28.458, 3.972, -37.923, -3.135]
  Set speed (120.0 mm/s)
  MoveL (T16313) to (105.67, 120.9, 17.7) mm, rotated rx 180 ry 0 rz -180 deg; joints [2.44, 66.314, -28.458, 3.972, -37.923, -3.135]
  Call Extruder -0.12811
  MoveL (T16314) to (105.93, 121.16, 17.7) mm, rotated rx 180 ry 0 rz -180 deg; joints [3.266, 68.593, -32.741, 5.565, -35.981, -4.508]
  Call Extruder -0.25189
  MoveL (T16315) to (105.22, 121.16, 17.7) mm, rotated rx 180 ry 0 rz -180 deg; joints [3.266, 68.593, -32.741, 5.565, -35.981, -4.508]
  Set speed (45.0 mm/s)
  Call Extruder -0.02
  MoveL (T16316) to (105.22, 121.16, 17.7) mm, rotated rx 180 ry 0 rz -180 deg; joints [3.266, 68.593, -32.741, 5.565, -35.981, -4.508]
  Set speed (150.0 mm/s)
  MoveL (T16317) to (105.22, 121.16, 19.7) mm, rotated rx 180 ry 0 rz -180 deg; joints [3.26, 68.907, -33.33, 5.591, -35.706, -4.545]
  MoveL (T16318) to (105.15, 117.23, 19.7) mm, rotated rx 180 ry 0 rz -180 deg; joints [3.26, 68.907, -33.33, 5.591, -35.706, -4.545]
  MoveL (T16319) to (105.15, 117.23, 17.7) mm, rotated rx 180 ry 0 rz -180 deg; joints [3.26, 68.907, -33.33, 5.591, -35.706, -4.545]
  Set speed (40.0 mm/s)
  Call Extruder 2.0
  MoveL (T16320) to (105.15, 117.23, 17.7) mm, rotated rx 180 ry 0 rz -180 deg; joints [2.362, 71.201, -37.642, 4.268, -33.632, -3.556]
  Set speed (50.0 mm/s)
  MoveL (T16321) to (105.15, 117.23, 17.7) mm, rotated rx 180 ry 0 rz -180 deg; joints [2.362, 71.201, -37.642, 4.268, -33.632, -3.556]
  Call Extruder 0.04143
  MoveL (T16322) to (105.15, 115.87, 17.7) mm, rotated rx 180 ry 0 rz -180 deg; joints [2.246, 71.187, -37.616, 4.057, -33.637, -3.379]
  Call Extruder 0.00661
  MoveL (T16323) to (105.23, 115.67, 17.7) mm, rotated rx 180 ry 0 rz -180 deg; joints [2.246, 71.187, -37.616, 4.057, -33.637, -3.379]
  Call Extruder 0.02637
  MoveL (T16324) to (105.84, 115.05, 17.7) mm, rotated rx 180 ry 0 rz -180 deg; joints [2.246, 71.187, -37.616, 4.057, -33.637, -3.379]
  Call Extruder 0.08606
  MoveL (T16325) to (103.84, 113.06, 17.7) mm, rotated rx 180 ry 0 rz -180 deg; joints [1.417, 68.707, -32.954, 2.424, -35.777, -1.967]
  Call Extruder 0.03385
  MoveL (T16326) to (103.84, 111.94, 17.7) mm, rotated rx 180 ry 0 rz -180 deg; joints [1.417, 68.707, -32.954, 2.424, -35.777, -1.967]
  Call Extruder 0.09463
  MoveL (T16327) to (106.04, 109.75, 17.7) mm, rotated rx 180 ry 0 rz -180 deg; joints [1.42, 68.396, -32.369, 2.413, -36.051, -1.951]
  Call Extruder 0.05062
  MoveL (T16328) to (105.29, 108.27, 17.7) mm, rotated rx 180 ry 0 rz -180 deg; joints [1.42, 68.396, -32.369, 2.413, -36.051, -1.951]
  Call Extruder 0.02377
  MoveL (T16329) to (105.1, 107.51, 17.7) mm, rotated rx 180 ry 0 rz -180 deg; joints [1.42, 68.396, -32.369, 2.413, -36.051, -1.951]
  Set speed (45.0 mm/s)
  Call Extruder -1.6
  MoveL (T16330) to (105.1, 107.51, 17.7) mm, rotated rx 180 ry 0 rz -180 deg; joints [2.319, 66.302, -28.436, 3.775, -37.927, -2.979]
  Set speed (120.0 mm/s)
  MoveL (T16331) to (105.1, 107.51, 17.7) mm, rotated rx 180 ry 0 rz -180 deg; joints [1.941, 66.269, -28.373, 3.158, -37.938, -2.491]
  Call Extruder -0.278
  MoveL (T16332) to (105.29, 108.27, 17.7) mm, rotated rx 180 ry 0 rz -180 deg; joints [1.941, 66.269, -28.373, 3.158, -37.938, -2.491]
  Call Extruder -0.102
  MoveL (T16333) to (105.42, 108.52, 17.7) mm, rotated rx 180 ry 0 rz -180 deg; joints [3.239, 69.919, -35.232, 5.678, -34.818, -4.667]
  Set speed (45.0 mm/s)
  Call Extruder -0.02
  MoveL (T16334) to (105.42, 108.52, 17.7) mm, rotated rx 180 ry 0 rz -180 deg; joints [3.239, 69.919, -35.232, 5.678, -34.818, -4.667]
  Set speed (150.0 mm/s)
  MoveL (T16335) to (105.42, 108.52, 19.7) mm, rotated rx 180 ry 0 rz -180 deg; joints [3.232, 70.25, -35.855, 5.708, -34.528, -4.708]
  MoveL (T16336) to (119.44, 110.51, 19.7) mm, rotated rx 180 ry 0 rz -180 deg; joints [3.232, 70.25, -35.855, 5.708, -34.528, -4.708]
  MoveL (T16337) to (119.44, 110.51, 17.7) mm, rotated rx 180 ry 0 rz -180 deg; joints [3.232, 70.25, -35.855, 5.708, -34.528, -4.708]
  Set speed (40.0 mm/s)
  Call Extruder 2.0
  MoveL (T16338) to (119.44, 110.51, 17.7) mm, rotated rx 180 ry 0 rz -180 deg; joints [3.232, 70.25, -35.855, 5.708, -34.528, -4.708]
  Set speed (50.0 mm/s)
  MoveL (T16339) to (119.44, 110.51, 17.7) mm, rotated rx 180 ry 0 rz -180 deg; joints [2.845, 71.266, -37.766, 5.145, -33.607, -4.289]
  Call Extruder 0.05098
  MoveL (T16340) to (118.25, 111.7, 17.7) mm, rotated rx 180 ry 0 rz -180 deg; joints [2.845, 71.266, -37.766, 5.145, -33.607, -4.289]
  Call Extruder 0.00661
  MoveL (T16341) to (118.05, 111.78, 17.7) mm, rotated rx 180 ry 0 rz -180 deg; joints [2.845, 71.266, -37.766, 5.145, -33.607, -4.289]
  Call Extruder 0.00686
  MoveL (T16342) to (117.83, 111.78, 17.7) mm, rotated rx 180 ry 0 rz -180 deg; joints [2.729, 71.249, -37.734, 4.933, -33.613, -4.112]
  Call Extruder 0.01607
